VAR_OUTPUT
	OUT_Error				: BOOL;
	OUT_Busy				: BOOL;
END_VAR

VAR
	ETAPE					: UINT;

    myStruct      			: ARRAY[1..CstNbLigneBuffer] OF St_DataHisto;
	myStructMax    			: ARRAY[1..CstNbLigneBufferMax] OF St_DataHisto;
	StructNull				: St_DataHisto;

    SQLDatabase				: FB_SQLDatabaseEvt('',T#10S);
	SQLCommand1				: FB_SQLCommandEvt('',T#10S);
	SQLCommandNull			: FB_SQLCommandEvt('',T#10S);
	bConnected				: BOOL;              	        	

	TrameValues				: T_MaxString := ' ([Timestamp],[Timestamp_Ms],[ParentId],[Value])';
	pPosRequete				: DINT;                		
	RequeteFinale			: ARRAY[1..100] OF STRING(1000);	
	RequeteFinaleNull		: ARRAY[1..100] OF STRING(1000);	
	sTimeStamp				: STRING(255);               	
	RequeteEntete			: STRING(1000);
	sInsertValue			: STRING(1000);
	Format					: FB_FormatString;
	                		
	NbElemBuffer			: DINT;
	KK						: DINT;
	                    	
	CmdStart				: BOOL;
	TrigCmdExec				: R_TRIG;
	TrigStart				: R_TRIG;
	RsStart					: RS;
	
	// Insert
		hDBID_BaseTampon	: UINT := 3;
	// AlarmManagement      
		bBufferMaxFull 		: BOOL;        		
		bInStructNull		: BOOL;
		
		
		
	
END_VAR

NbElemBuffer := M_Count();
CmdStart := NbElemBuffer>= CstNbLigneBuffer;


TrigStart(CLK := CmdStart);
IF TrigStart.Q THEN
	FOR KK := 1 TO CstNbLigneBuffer DO
		myStruct[KK] := myStructMax[KK];
	END_FOR
END_IF


// call functionblock

CASE ETAPE OF
	0://INITIALISATION  & CONNECTION
		RequeteEntete := concat(concat('INSERT INTO ',NomTable),concat(TrameValues,' VALUES '));
		RsStart(SET := TrigStart.Q);
		IF RsStart.Q1 THEN
			IF SQLDatabase.Connect(hDBID := hDBID) THEN;
				bConnected := NOT sqldatabase.bError;
				IF bConnected THEN
					ETAPE := 1;
				ELSE
					ETAPE := 255;
				END_IF
			END_IF
		END_IF
		
	1: // CONNECTED
		IF SQLDatabase.CreateCmd(pSQLCommand := ADR(SQLCommand1)) THEN 
			IF NOT SQLCommand1.bError THEN
				ETAPE := 2;
			ELSIF SQLCommand1.bError THEN
				ETAPE := 255;
			END_IF
		END_IF
	2:
		MEMCPY(srcAddr:= ADR(RequeteEntete), destAddr := ADR(requeteFinale), n:= SIZEOF(RequeteEntete));
		pPosRequete := LEN(STR := RequeteEntete);
		FOR KK:= 1 TO CstNbLigneBuffer-1 DO
			sTimeStamp	:= right(STR := DT_TO_STRING(myStruct[KK].Timestamp), SIZE := LEN(DT_TO_STRING(myStruct[KK].Timestamp))-3);
			Format(sFormat := '($'%s $',%.3d,%.4d,%5.2f),', arg1 := F_STRING(sTimeStamp),arg2:=F_DINT(myStruct[KK].Timestamp_Ms), arg3:= F_DINT(myStruct[KK].ParentId), arg4:= F_LREAL(myStruct[KK].Value), sOut=>sInsertValue);
			MEMCPY(srcAddr:= ADR(sInsertValue), destAddr := ADR(requeteFinale)+DINT_TO_DWORD(pPosRequete), n:= SIZEOF(sInsertValue));
			pPosRequete:= pPosRequete + LEN(STR := sInsertValue);
		END_FOR
		sTimeStamp	:= right(STR := DT_TO_STRING(myStruct[KK].Timestamp), SIZE := LEN(DT_TO_STRING(myStruct[KK].Timestamp))-3);
		Format(sFormat := '($'%s $',%.3d,%.4d,%5.2f)', arg1 := F_STRING(sTimeStamp),arg2:=F_DINT(myStruct[KK].Timestamp_Ms), arg3:= F_DINT(myStruct[KK].ParentId), arg4:= F_LREAL(myStruct[KK].Value), sOut=>sInsertValue);
		MEMCPY(srcAddr:= ADR(sInsertValue), destAddr := ADR(requeteFinale)+DINT_TO_DWORD(pPosRequete), n:= SIZEOF(sInsertValue));
	
		IF SQLCommand1.Execute(pSQLCmd := ADR(RequeteFinale), cbSQLCmd := SIZEOF(Requetefinale))THEN
			
			IF  NOT SQLCommand1.bError THEN
				ETAPE := 3;
			ELSIF SQLCommand1.bError THEN
				ETAPE := 255;
			END_IF
		END_IF
	3:
			IF SQLDatabase.Disconnect() THEN
				ETAPE := 4;
			END_IF 
	4:
		IF NOT SQLDatabase.bError THEN
			RequeteFinale := RequeteFinaleNull;
			FOR KK := CstNbLigneBuffer TO CstNbLigneBufferMax -1 DO
				myStructMax[KK+1-CstNbLigneBuffer]:= myStructMax[KK+1];
			END_FOR
			
			FOR KK := CstNbLigneBufferMax-CstNbLigneBuffer+1 TO CstNbLigneBufferMax DO
				myStructMax[KK]:= StructNull;
			END_FOR			
			
			TrigStart(CLK := FALSE);
			RsStart(RESET1 := TRUE);
			RsStart(RESET1 := FALSE);
			TrigCmdExec(CLK := FALSE);
			CmdStart := FALSE;
			Etape := 0;
			OUT_Error := FALSE;
		ELSE 
			ETAPE := 255;
		END_IF
	255: 
		RequeteFinale := RequeteFinaleNull;
		OUT_Error := TRUE;
		Etape := 0;
		RsStart(RESET1 := TRUE);
		RsStart(RESET1 := FALSE);
		TrigCmdExec(CLK := FALSE);
		CmdStart := FALSE;
		
END_CASE

METHOD M_AddLine : BOOL
VAR_INPUT
	InStruct			: St_DataHisto;
END_VAR

VAR
END_VAR
// Check the biggest buffer isn't full
IF MEMCMP(pBuf1 := ADR(StructNull), pBuf2 := ADR(myStructMax[CstNbLigneBufferMax]), n := SIZEOF(StructNull)) <> 0 THEN
	bBufferMaxFull := TRUE;
ELSE
	//Check the input struct isn't null
	IF MEMCMP(pBuf1 := ADR(StructNull), pBuf2 := ADR(InStruct), n := SIZEOF(StructNull)) = 0 THEN
		bInStructNull := TRUE;
	ELSE
		// We parse the biggest buffer
		FOR KK := 1 TO CstNbLigneBufferMax DO 
			IF MEMCMP(pBuf1 := ADR(StructNull), pBuf2 := ADR(myStructMax[KK]), n := SIZEOF(StructNull)) = 0 THEN
				myStructMax[KK] := InStruct;
				bBufferMaxFull := FALSE;
				EXIT;
			END_IF
		END_FOR
	END_IF
END_IF
END_METHOD

METHOD M_AlarmManager : BOOL
VAR_INPUT
	AlarmCode : WORD;
	
END_VAR


AlarmCode.0 := bBufferMaxFull;
AlarmCode.1 := bInStructNull;
END_METHOD

METHOD M_Count : DINT
VAR_INPUT
END_VAR
VAR

END_VAR
FOR KK := 1 TO CstNbLigneBufferMax DO 

	IF MEMCMP(pBuf1 := ADR(StructNull), pBuf2 := ADR(myStructMax[KK]), n := SIZEOF(StructNull)) = 0 THEN
		EXIT ;
	END_IF
END_FOR

M_Count := MIN(KK, CstNbLigneBufferMax);
END_METHOD

END_FUNCTION_BLOCK

// ---- 00_FunctionsBlocks/Database/SQLite/SQLite_CreateDb_V2_1.TcPOU
PROGRAM SQLite_CreateDb_V2_1
VAR_INPUT
	IN_ConfigDbActuelle		: ARRAY[0..MAX_CONFIGURATIONS] OF ST_ConfigDB; 
	IN_DbType				: UINT:= 1; // 1:T_DBConfig_SQLite, 2:T_DBConfig_SQLCe
	IN_Dir					: T_MAXSTRING;
	IN_Name					: STRING;
	IN_Start				: BOOL;
	IN_TableName			: STRING;
END_VAR
VAR_IN_OUT
	IN_hDBID         		: UDINT;	
END_VAR
VAR_OUTPUT
	OUT_Error				: BOOL;
	OUT_Busy				: BOOL;
	OUT_Result				: INT;
END_VAR
VAR
	Etape					: UINT;
	
	TrigStart				: R_TRIG;
	RsStart					: RS;
	bCreateTable			: BOOL;
	TrigCreateTable			: R_TRIG;
	RsCreateTable			: RS;
	PLCDBCreateEvt 			: FB_PLCDBCreateEvt(sNetID := '', tTimeout := T#5S);
	SqlLiteConf				: T_DBConfig_SQLite;
	DbFullDirName			: T_MAXSTRING;	
	sExtension				: STRING:= '.db';
	tcMessage    	 		: I_TcMessage;
	
	AX_ColArray				: ARRAY[0..3] OF ST_ColumnInfo;
	
	dBID_Test				: UDINT := 1;
	KK						: UDINT;
	bExisteDeja				: BOOL;	
END_VAR

OUT_Busy := TRUE;
AX_ColArray[0].sName := 'TimeStamp';     	AX_ColArray[0].eType := E_ColumnType.DateTime;   	AX_ColArray[0].nLength := 4;    
AX_ColArray[1].sName := 'TimeStamp_Ms';    	AX_ColArray[1].eType := E_ColumnType.Integer;    	AX_ColArray[1].nLength := 4;
AX_ColArray[2].sName := 'ParentId';   		AX_ColArray[2].eType := E_ColumnType.Integer;   	AX_ColArray[2].nLength := 4;
AX_ColArray[3].sName := 'Value';   			AX_ColArray[3].eType := E_ColumnType.Float;   		AX_ColArray[3].nLength := 8;


IF IN_DbType = 1 THEN
	sExtension := '.db';
ELSIF IN_DbType = 2 THEN
	sExtension := '.sdf';
END_IF

DbFullDirName := Concat(STR1:=Concat(STR1:= IN_Dir, STR2 := IN_Name), STR2 := sExtension);
SqlLiteConf.bAuthentification := FALSE;
SqlLiteConf.sServer := DbFullDirName;

FOR KK := 0 TO MAX_CONFIGURATIONS DO
	IF IN_ConfigDbActuelle[KK].sServer = DbFullDirName THEN
		bExisteDeja := TRUE;
		OUT_Result := -1;
		OUT_Busy := FALSE;
		OUT_Error := FALSE;
		bCreateTable := FALSE;
		IN_hDBID := IN_ConfigDbActuelle[KK].hDBID;
		EXIT;
	END_IF
	IF KK = MAX_CONFIGURATIONS THEN
		bExisteDeja := FALSE;
	END_IF
END_FOR

TrigStart(CLK := IN_Start AND NOT bExisteDeja);
RsStart(SET := TrigStart.Q);
IF RsStart.Q1 THEN
	IF PLCDBCreateEvt.Database(pDatabaseConfig := ADR(SqlLiteConf), cbDatabaseConfig := SIZEOF(SqlLiteConf), bCreateXMLConfig := TRUE, pDBID := ADR(dBID_Test)) THEN
		IF PLCDBCreateEvt.ipTcResult.nEventId = 59 THEN
			OUT_Error := FALSE;
			OUT_Result := -1;
			OUT_Busy := FALSE;	
			TrigStart(CLK := FALSE);
			bCreateTable := FALSE;
			Etape := 0;
			RsCreateTable(RESET1 := TRUE);
			RsCreateTable(RESET1 := FALSE);
		ELSIF PLCDBCreateEvt.bError THEN
			tcMessage := PLCDBCreateEvt.ipTcResult;
			OUT_Error := TRUE;
		ELSE
			Etape := 1;
			IN_hDBID := dBID_Test;
			bCreateTable := TRUE; 
		END_IF
		RsStart(RESET1 := TRUE);
		RsStart(RESET1 := FALSE);
	END_IF
END_IF

TrigCreateTable(CLK := bCreateTable);
RsCreateTable(SET:= TrigCreateTable.Q);

IF RsCreateTable.Q1 AND ETAPE = 1 THEN
	IF PLCDBCreateEvt.Table(hDBID := IN_hDBID, sTableName := IN_TableName,  pTableCfg := ADR(AX_ColArray), cbTableCfg := SIZEOF(AX_ColArray)  ) THEN
		IF PLCDBCreateEvt.bError THEN
			Etape := 255;
			OUT_Error := TRUE;
			OUT_Result := -2;
		ELSE
			IN_Start := FALSE;
			bCreateTable := FALSE;
			Etape := 0;
			OUT_Result := 1;
			RsCreateTable(RESET1 := TRUE);
			RsCreateTable(RESET1 := FALSE);
			TrigStart(CLK := False);
			OUT_Busy := FALSE;	
			OUT_Error := FALSE;
		END_IF
	END_IF
END_IF

IF Etape = 255 THEN
	Etape := 0;
	bCreateTable := FALSE;
	IN_Start := FALSE;
	OUT_Busy := FALSE;	
	RsCreateTable(RESET1 := TRUE);
	RsCreateTable(RESET1 := FALSE);
	
END_IF

END_PROGRAM

// ---- 00_FunctionsBlocks/Database/SQLite/SQLite_DeleteConfDb_1.TcPOU
PROGRAM SQLite_DeleteConfDb_1
VAR_INPUT
	IN_DbType				: UINT:= 1; // 1:T_DBConfig_SQLite, 2:T_DBConfig_SQLCe
	IN_hDBID         		: UDINT;
	IN_Start				: BOOL;
	
END_VAR
VAR_OUTPUT
	OUT_Error				: BOOL;
	OUT_Busy				: BOOL;
END_VAR
VAR
	Etape					: UINT;
	
	TrigStart				: R_TRIG;
	RsStart					: RS;
	bDeleteTable			: BOOL;
	TrigDeleteFile			: R_TRIG;
	RsDeleteTable			: RS;
	fbConfigTcDBSrv   		: FB_ConfigTcDBSrvEvt (sNetID := '', tTimeout := T#5S);
	DbFullDirName			: T_MAXSTRING;	
	sExtension				: STRING:= '.db';
	tcMessage    	 		: I_TcMessage;
	
	

END_VAR

OUT_Busy := TRUE;

TrigStart(CLK := IN_Start);
RsStart(SET := TrigStart.Q);
IF RsStart.Q1 THEN
	IF fbConfigTcDBSrv.Delete(eTcDBSrvConfigType := E_TcDBSrvConfigType.Database, hConfigID := IN_hDBID) THEN
		IF fbConfigTcDBSrv.bError THEN
			tcMessage := fbConfigTcDBSrv.ipTcResult;
			OUT_Error := TRUE;
			OUT_Busy := FALSE;
			Etape := 255;
		ELSE 
			OUT_Busy := FALSE;
			OUT_Error := FALSE;
			Etape := 0;
		END_IF
		TrigStart(CLK := FALSE);
		RsStart(RESET1 := TRUE);
		RsStart(RESET1 := FALSE);
	END_IF
END_IF

IF Etape = 255 THEN
	Etape := 0;
	bDeleteTable := FALSE;
	IN_Start := FALSE;
	OUT_Busy := FALSE;	
	RsDeleteTable(RESET1 := TRUE);
	RsDeleteTable(RESET1 := FALSE);
	
END_IF

END_PROGRAM

// ---- 00_FunctionsBlocks/Database/UnixTimestamp.TcPOU
FUNCTION_BLOCK UnixTimestamp
VAR_OUTPUT
    seconds: ULINT;
    milliseconds: ULINT;
END_VAR

VAR
    localSystemTime : FB_LocalSystemTime := ( bEnable := TRUE, dwCycle := 1 );
    getTimeZoneInformation : FB_GetTimeZoneInformation;
    timeZoneInformation : ST_TimeZoneInformation;
    specificLocalTimeToFileTime : FB_TzSpecificLocalTimeToFileTime;
    fileTime: T_FILETIME;
    onZerothSecondLastCycle : BOOL;
END_VAR

// Get local system time
localSystemTime();

// On the zeroth second of each minutesync timezone information
IF (timeZoneInformation.standardName = '' OR (localSystemTime.systemTime.wSecond = 0 AND NOT onZerothSecondLastCycle)) THEN
    getTimeZoneInformation(sNetID := '', bExecute := TRUE, tzInfo => timeZoneInformation);
END_IF;

// Convert local system time to unix timestamps
specificLocalTimeToFileTime(in := Tc2_Utilities.SYSTEMTIME_TO_FILETIME(localSystemTime.systemTime), tzInfo := timeZoneInformation, out => fileTime);
seconds := (SHL(DWORD_TO_ULINT(fileTime.dwHighDateTime), 32) + DWORD_TO_ULINT(fileTime.dwLowDateTime)) / 10000000 - 11644473600;
milliseconds := (SHL(DWORD_TO_ULINT(fileTime.dwHighDateTime), 32) + DWORD_TO_ULINT(fileTime.dwLowDateTime)) / 10000 - 11644473600000;

onZerothSecondLastCycle := localSystemTime.systemTime.wSecond = 0;

END_FUNCTION_BLOCK

// ---- 00_FunctionsBlocks/DataProcessing/Compress/FB_CompressFile.TcPOU
FUNCTION_BLOCK FB_CompressFile
// FB to Compress all files of the directory. 
VAR_INPUT
	IN_Directory			: T_MaxString; // directory of the file to compress
END_VAR
VAR_OUTPUT
END_VAR
VAR
	StartProcess 			: NT_StartProcess;
	bTest 					: BOOL;
	TrigJour				: R_TRIG;
	RsJour					: RS;
	DirAlarms				: T_MaxString;
	DirRawdata				: T_MaxString;
	TimeStructYesterday		: TIMESTRUCT;
END_VAR


TrigJour(CLK := CalLocalTimeStruct.wHour =0);
RsJour(SET := TrigJour.Q);

TimeStructYesterday := DT_TO_SYSTEMTIME( SYSTEMTIME_TO_DT (CalLocalTimeStruct) - T#1D);

IF RsJour.Q1 THEN
	DirAlarms := CONCAT(STR1 := CONCAT(STR1 := CONCAT(STR1 := CONCAT(STR1 := CONCAT(STR1 := CONCAT(STR1 := CONCAT(STR1 := CONCAT(STR1 := CONCAT(STR1 := Concat(STR1 := Concat(STR1 := IN_Directory, STR2 := WORD_TO_STRING(TimeStructYesterday.wYear)), STR2 := '\'), STR2 := WORD_TO_STRING(TimeStructYesterday.wMonth)), STR2 := '\'), STR2:='ALARMS_'), STR2:= WORD_TO_STRING(TimeStructYesterday.wYear)), STR2:='-'),STR2:=WORD_TO_STRING(TimeStructYesterday.wMonth)),STR2:='-'),STR2:=WORD_TO_STRING(TimeStructYesterday.wDay)),STR2:='.csv');
	DirRawdata:= CONCAT(STR1 := CONCAT(STR1 := CONCAT(STR1 := CONCAT(STR1 := CONCAT(STR1 := CONCAT(STR1 := CONCAT(STR1 := CONCAT(STR1 := CONCAT(STR1 := Concat(STR1 := Concat(STR1 := IN_Directory, STR2 := WORD_TO_STRING(TimeStructYesterday.wYear)), STR2 := '\'), STR2 := WORD_TO_STRING(TimeStructYesterday.wMonth)), STR2 := '\'), STR2:='RAWDATA_'), STR2:= WORD_TO_STRING(TimeStructYesterday.wYear)), STR2:='-'),STR2:=WORD_TO_STRING(TimeStructYesterday.wMonth)),STR2:='-'),STR2:=WORD_TO_STRING(TimeStructYesterday.wDay)),STR2:='.csv');
	StartProcess
	(
		NETID := '',
		PATHSTR := 'C:\Windows\System32\compact.exe',
		DIRNAME := 'C:\Windows\System32',
		COMNDLINE :=  CONCAT(STR1:=CONCAT(STR1:=CONCAT(STR1:=CONCAT(STR1:=' /c "',STR2:=DirAlarms), str2:='"  "'), STR2:=DirRawdata),str2:='"'),
		Start := RsJour.Q1,
		TMOUT := T#3M
	);
	IF NOT StartProcess.BUSY THEN
		IF NOT StartProcess.ERR THEN
			StartProcess(Start := FALSE);
			RsJour(RESET1:= TRUE);
			RsJour(RESET1:= FALSE);
		ELSE
			StartProcess(Start := FALSE);
		END_IF
	END_IF	
END_IF

END_FUNCTION_BLOCK

// ---- 00_FunctionsBlocks/DataProcessing/Compress/FUN_CompressCSV.TcPOU
PROGRAM FUN_CompressCSV
VAR_INPUT
	InDirectory 		: T_MaxString;
END_VAR
VAR_OUTPUT
END_VAR
VAR
	Directory1		: T_MaxString;
	Directory2		: T_MaxString;
	FB_Time 			: FB_LocalSystemTime;
	CompressFile	: FB_CompressFile;
	PreviousMonth 	: WORD := 12;
	PreviousYear 	: WORD := 2018;
	CalDirectory 	: T_MaxString;
	DirChange		: BOOL;
	bTest 			: BOOL;
	TimeStruct_Local : TIMESTRUCT;
END_VAR

FB_Time(sNetID := '', bEnable := TRUE, dwCycle := 1, dwOpt := 1, tTimeout := T#50MS, systemTime => TimeStruct_Local);
IF FB_TIME.bValid THEN 
	IF PreviousMonth <> TimeStruct_Local.wMonth THEN
		Directory1 := Concat(InDirectory, concat(WORD_TO_STRING(TimeStruct_Local.wYear), '\'));
		
		IF PreviousYear <> TimeStruct_Local.wYear THEN
			Directory1 := Concat(InDirectory, concat(WORD_TO_STRING(TimeStruct_Local.wYear-1), '\'));
			PreviousYear := TimeStruct_Local.wYear;
		END_IF
		
		Directory2 := Concat(Directory1, concat(WORD_TO_STRING(PreviousMonth), '\'));
		PreviousMonth := TimeStruct_Local.wMonth;
		DirChange := TRUE;
	END_IF

	
	IF DirChange THEN	
		bTest := TRUE;
		CompressFile(IN_Directory := Directory2);	
		DirChange := FALSE;
	END_IF
END_IF

END_PROGRAM

// ---- 00_FunctionsBlocks/DataProcessing/Database/DataBase_V2.TcPOU
PROGRAM DataBase_V2
// Cette fois, plutôt qu'1 base avec 3 tables, faire 3 bases par jour (100ms, 1s, 1m)
// Nouvelle architecture : fichiers minute dans le même fichier qu'historisation, les autres dans Database
 
VAR
	ParamBaseDir					: T_MAXString := 'C:\TwinCAT\Functions\Database\SQLite\';
	ParamHistDir					: T_MaxString := 'C:\TwinCAT\Functions\Historisation\';
	
	ParamDbType						: UINT;
	                        		
	DBID_GLOBAL						: ARRAY[1..3] OF UDINT;
	DBID_ToDelete					: ARRAY[1..3] OF UDINT;
	
	bTest							: BOOL;
	
    AX_DirDB						: ARRAY[1..3] OF T_MaxString :=[ParamBaseDir, ParamBaseDir, ParamBaseDir] ;
	                   		
	MesAlarmCode 					: WORD;
	MesWarningCode					: WORD;
	// INIT
		
                            		
	// CheckConfig          		
		bCheckConfig				: BOOL := TRUE;
		TrigCheckConfig				: R_TRIG;
		TrigInit					: F_TRIG;
		RS_CheckConfig				: RS;
		                    		
		ConfigTcDBSrvEvt  			: FB_ConfigTcDBSrvEvt(sNetId := '', tTimeout:=T#5S);
		                    		
		aDBConfig         			: ARRAY[0..MAX_CONFIGURATIONS] OF ST_ConfigDB;
		aAutoGrpConfig    			: ARRAY[0..MAX_CONFIGURATIONS] OF ST_ConfigAutoLogGrp;
		AX_NameBase					: ARRAY[0..MAX_CONFIGURATIONS] OF T_MaxString;
		AX_hDBID					: ARRAY[0..MAX_CONFIGURATIONS] OF BOOL;
		AX_hDBIDNull				: ARRAY[0..MAX_CONFIGURATIONS] OF BOOL;
		                    		
		nDbCount          			: UDINT;
		nAutoGrpCount     			: UDINT;
		tcMessage         			: I_TcMessage;
	
	// DayTrig 
		Trig_CreateFolder			: R_TRIG;
		RS_CreateFolder				: RS;
		RS_CreateDbDay				: RS;
		RS_DeleteConf				: RS;
		RS_DeleteFiles				: RS;
		RS_CompressOldFiles			: RS;
		bDayTrig					: BOOL:= TRUE;
		bCreateDirErr				: BOOL;
		bCreateDbErr				: BOOL;
		bDeleteConfErr				: BOOL;
		bDeleteFileErr				: BOOL;
		bCompressFileErr			: BOOL;
		CreateDir					: FB_CreateDir_V2;
        AX_Name						: ARRAY[1..3] OF STRING;    
		DeleteFile30Days			: FB_DeleteFile;          
		DeleteFile3Days				: FB_DeleteFile;          
		StartProcess 				: NT_StartProcess;
		
	// CreateDb Init        		
		bCreateDb					: BOOL := TRUE;
		DbidCreated					: UDINT := 1;
		DbCreated_Trig				: F_TRIG;
		AX_ColArray					: ARRAY[0..3] OF ST_ColumnInfo;
	                            	
	// One hour has elapsed
		Trig1hour					: R_TRIG;
		Rs1hour						: RS;
		OldDBID						: UDINT := 1;
		bDbCreated					: BOOL;
		bDbDelete					: BOOL;
		sReqCmd						: T_MAXSTRING;
		
	// New day 
		TrigJour					: R_TRIG;
		RsJour						: RS;
		b1jourSpDoing				: BOOL;
		TimeStruct3days				: TIMESTRUCT;
		TimeStruct1month			: TIMESTRUCT;
		Requete						: T_MaxString;
		sTimeStamp1					: STRING(255);
		sTimeStamp2					: STRING(255);
		Format						: FB_FormatString;
	
		
	// Insert	
	SQLExpert_InsertBuffer_1s		: FB_SQLExpert_InsertBuffer;
	SQLExpert_InsertBuffer_1m		: FB_SQLExpert_InsertBuffer;
	SQLExpert_InsertBuffer_100ms	: FB_SQLExpert_InsertBuffer;

	TON_100ms						: TON;
	TON_1m							: TON;
	TON_1s							: TON;
	

	
	bInit 							: BOOL := TRUE;
	KK								: UDINT;
	LL								: UDINT := 1;

	bTest1 							: BOOL;
	bTest2 							: BOOL;
	
END_VAR

// Trigger pour détecter nouvelle journée -> lance un check config + DayTrig pour faire les proc stockées
TrigJour(CLK := CalLocalTimeStruct.wHour = 0);
bCheckConfig := TrigJour.Q;
Trig_CreateFolder(CLK := TrigJour.Q OR binit);
RS_CreateFolder(SET := Trig_CreateFolder.Q);

// Methode pour vérifier la configuration actuellement activée sur front montant de bCheckConfig
M_Checkconfig();

IF NOT bCheckConfig THEN
	M_DayTrig();
END_IF 

IF bInit THEN
	M_Init();
END_IF

M_AlarmManagement();
(*--------------------------------------------------------------------------------------------*)
(*--------------------------------------------------------------------------------------------*)
// ICI JE LANCE LES ADD BUFFER POUR LES 3 TABLES
IF NOT bInit THEN
	SQLExpert_InsertBuffer_100ms(NomTable := 'Table100ms', hDBID := DBID_GLOBAL[1]);
	SQLExpert_InsertBuffer_1s(NomTable := 'Table1s', hDBID := DBID_GLOBAL[2]);
	SQLExpert_InsertBuffer_1m(NomTable := 'Table1m', hDBID := DBID_GLOBAL[3]);
	
	
	TON_100ms(IN := NOT bInit, PT := T#100MS);
	IF TON_100ms.Q THEN
		FOR KK := 1 TO 100 DO
			SQLExpert_InsertBuffer_100ms.M_AddLine(InStruct := GVL_DataBaseStructures.AX_Struct_100ms[KK]);
		END_FOR
		TON_100ms(IN := FALSE);
		TON_100ms(IN := TRUE);
	END_IF
	
	TON_1s(IN := NOT bInit, PT := T#1S);
	IF TON_1s.Q THEN
		FOR KK := 1 TO 1000 DO
			SQLExpert_InsertBuffer_1s.M_AddLine(InStruct := GVL_DataBaseStructures.AX_Struct_1s[KK]);
		END_FOR
		TON_1s(IN := FALSE);
		TON_1s(IN := TRUE);
	END_IF
	
	TON_1m(IN := NOT bInit, PT := T#1M);
	IF TON_1m.Q THEN
		FOR KK := 1 TO 1000 DO
			SQLExpert_InsertBuffer_1m.M_AddLine(InStruct := GVL_DataBaseStructures.AX_Struct_1m[KK]);
		END_FOR
		TON_1m(IN := FALSE);
		TON_1m(IN := TRUE);
	END_IF	

END_IF
(*--------------------------------------------------------------------------------------------*)
(*--------------------------------------------------------------------------------------------*)

METHOD M_AlarmManagement : BOOL
VAR
		FB_AlarmCodeManager : FB_AlarmCodeManager;
END_VAR
FB_AlarmCodeManager
(
	bAlarm1 := bCreateDirErr,
	bAlarm2 := bCreateDbErr,
	bAlarm3 := bDeleteConfErr,
	bAlarm4 := bDeleteFileErr,
	bAlarm5 := bCompressFileErr,
	wAlarmCode => MesAlarmCode
);
END_METHOD

METHOD M_CheckConfig : BOOL
VAR_INPUT
END_VAR
TrigCheckConfig(CLK := bCheckConfig OR binit);
RS_CheckConfig(SET := TrigCheckConfig.Q);
	
IF RS_CheckConfig.Q1 THEN
	IF ConfigTcDBSrvEvt.Read(
		pDBConfig := ADR(aDBConfig), 
		cbDBConfig := SIZEOF(aDBConfig), 
		pAutologGrpConfig := ADR(aAutoGrpConfig),
		cbAutoLogGrpConfig := SIZEOF(aAutoGrpConfig),
		pDBCount := ADR(nDbCount),
		pAutoLogGrpCount := ADR(nAutoGrpCount))
	 THEN
		IF ConfigTcDBSrvEvt.bError THEN
			tcMessage := ConfigTcDBSrvEvt.ipTcResult;
			bCheckConfig := FALSE; 
		ELSE
			bCheckConfig := FALSE; 
			FOR KK := 0 TO MAX_CONFIGURATIONS DO
				AX_hDBID[aDBConfig[KK].hDBID] := aDBConfig[KK].hDBID <> 0;
				AX_NameBase[KK] :=  aDBConfig[KK].sName;
			END_FOR
		END_IF  
		TrigCheckConfig(CLK := FALSE OR binit);
		RS_CheckConfig(RESET1 := TRUE);
		RS_CheckConfig(RESET1 := FALSE);
	END_IF
END_IF
END_METHOD

METHOD M_DayTrig : BOOL
VAR_INPUT
END_VAR
VAR
	DirTemp			: ARRAY[1..3] OF T_MaxString;
	AX_NameTemp		: ARRAY[1..3] OF STRING := ['Table100ms', 'Table1s', 'Table1m']; 	
	Dir30Days		: T_MaxString;
	Dir3Days		: T_MaxString; 	
	Dir3DaysComp1	: T_MaxString; 	
	Dir3DaysComp2	: T_MaxString; 	

	
END_VAR



TimeStruct3days := DT_TO_SYSTEMTIME( SYSTEMTIME_TO_DT (CalLocalTimeStruct) - T#3D);
TimeStruct1month := DT_TO_SYSTEMTIME( SYSTEMTIME_TO_DT (CalLocalTimeStruct) - T#30D);

// D'abord je commence par créer tous les dossiers
IF RS_CreateFolder.Q1 THEN
	DirTemp[1] := ParamHistDir;
	DirTemp[2] := Concat(STR1 := Concat(STR1 := ParamHistDir, STR2 := WORD_TO_STRING(CalLocalTimeStruct.wYear)), STR2 := '\');
	DirTemp[3] := CONCAT(STR1 := CONCAT(STR1 := Concat(STR1 := Concat(STR1 := ParamHistDir, STR2 := WORD_TO_STRING(CalLocalTimeStruct.wYear)), STR2 := '\'), STR2 := WORD_TO_STRING(CalLocalTimeStruct.wMonth)), STR2 := '\');
	
	AX_DirDB[1] := ParamBaseDir;
	AX_DirDB[2] := ParamBaseDir;
	AX_DirDB[3] := DirTemp[3];
	FOR KK := 1 TO 3 DO 
		AX_Name[KK] := CONCAT(STR1 := CONCAT(STR1 := CONCAT(STR1 := CONCAT(STR1 := CONCAT(STR1 := Concat(STR1 := WORD_TO_STRING(CalLocalTimeStruct.wYear), STR2 := ''), STR2 := WORD_TO_STRING(CalLocalTimeStruct.wMonth)), STR2:= ''), STR2:= WORD_TO_STRING(CalLocalTimeStruct.wDay)), STR2:= '_'), STR2:= AX_NameTemp[KK]);
	END_FOR
	
	IF LL < 4 THEN
		CreateDir(InPath := DirTemp[LL], InExe := LL < 4);
		IF NOT CreateDir.OutBusy THEN
			IF CreateDir.OutError AND NOT CreateDir.OutErrorId =1827 (*Dossier existe déjà*) THEN
				CreateDir(InExe := FALSE);
				bCreateDirErr := TRUE;
			ELSE
				bCreateDirErr := FALSE;
				CreateDir(InExe := FALSE);
				LL := LL + 1;
			END_IF
			CreateDir(InPath := DirTemp[LL], InExe := FALSE);
		END_IF
	ELSE
		RS_CreateFolder(RESET1 := TRUE);
		RS_CreateFolder(RESET1 := FALSE);
		RS_CreateDbDay(SET := TRUE);
		RS_CreateDbDay(SET := FALSE);
		LL := 1;
	END_IF
END_IF

// Ensuite je créée les bases 
IF RS_CreateDbDay.Q1 THEN
	IF LL < 4 THEN
		SQLite_CreateDb_V2(IN_DbType := 1, IN_Dir := AX_DirDB[LL],IN_Name := AX_Name[LL], IN_TableName := AX_NameTemp[LL], IN_hDBID := DBID_GLOBAL[LL], IN_Start := bCreateDb, IN_ConfigDbActuelle := aDBConfig);
		IF NOT SQLite_CreateDb_V2.OUT_Busy THEN
			SQLite_CreateDb_V2(IN_Start := FALSE, IN_hDBID := DBID_GLOBAL[LL]);
			IF SQLite_CreateDb_V2.OUT_Error THEN
				SQLite_CreateDb_V2(IN_Start := FALSE, IN_hDBID := DBID_GLOBAL[LL]);
				bCreateDbErr := TRUE;
			ELSE
				SQLite_CreateDb_V2(IN_Start := FALSE, IN_hDBID := DBID_GLOBAL[LL]);
				LL := LL + 1;
				bCreateDbErr := FALSE;
			END_IF
		END_IF
	ELSE
		LL := 1;
		RS_CreateDbDay(RESET1 := TRUE);
		RS_CreateDbDay(RESET1 := FALSE);
		RS_DeleteConf(SET := TRUE AND NOT bInit);
		RS_DeleteConf(SET := FALSE);
		bDayTrig := False;
	END_IF
END_IF

// Ensuite je supprime les vieilles tables de la conf précédente
IF RS_DeleteConf.Q1 THEN
	IF LL < 4 THEN
		DBID_ToDelete[LL] := SEL(DBID_GLOBAL[LL] = LL, LL, LL+3);
		// CELA NE SUPPRIME QUE LES CONFS
		SQLite_DeleteConfDb(IN_DbType := 1, IN_hDBID := DBID_ToDelete[LL], IN_Start := TRUE);
		IF NOT SQLite_DeleteConfDb.OUT_Busy THEN
			IF SQLite_DeleteConfDb.OUT_Error THEN
				SQLite_DeleteConfDb(IN_Start := FALSE);
				bDeleteConfErr := TRUE;
			ELSE
				bDeleteConfErr := FALSE;
				SQLite_DeleteConfDb(IN_Start := FALSE);
				LL := LL + 1;
			END_IF
		END_IF
	ELSE
		LL := 1;
		RS_DeleteConf(RESET1 := TRUE);
		RS_DeleteConf(RESET1 := FALSE);
		RS_DeleteFiles(SET := TRUE);
		RS_DeleteFiles(SET := FALSE);
	END_IF
END_IF

// Et enfin, je supprime les vieux fichiers : plus de 30 jours pour les 1s, plus de 3 jours pour les 100ms
IF RS_DeleteFiles.Q1 THEN
	Dir30Days := CONCAT(STR1:=CONCAT(STR1:=CONCAT(STR1 := CONCAT(STR1 := CONCAT(STR1 := CONCAT(STR1 := CONCAT(STR1 := Concat(STR1 := ParamBaseDir, STR2 := WORD_TO_STRING(TimeStruct1month.wYear)), STR2 := ''), STR2 := WORD_TO_STRING(TimeStruct1month.wMonth)), STR2:= ''), STR2:= WORD_TO_STRING(TimeStruct1month.wDay)), STR2:= '_'), STR2:= AX_NameTemp[LL]), STR2 := '.db');
	Dir3Days := CONCAT(STR1:=CONCAT(STR1:=CONCAT(STR1 := CONCAT(STR1 := CONCAT(STR1 := CONCAT(STR1 := CONCAT(STR1 := Concat(STR1 := ParamBaseDir, STR2 := WORD_TO_STRING(TimeStruct3days.wYear)), STR2 := ''), STR2 := WORD_TO_STRING(TimeStruct3days.wMonth)), STR2:= ''), STR2:= WORD_TO_STRING(TimeStruct3days.wDay)), STR2:= '_'), STR2:= AX_NameTemp[LL]), STR2 := '.db');
	
	DeleteFile30Days(IN_Dir := Dir30Days, IN_Start := TRUE);
	DeleteFile3Days(IN_Dir := Dir3Days, IN_Start := TRUE);
	
	IF NOT DeleteFile3Days.OUT_Busy AND NOT DeleteFile30Days.OUT_Busy AND LL < 2 THEN
		IF NOT DeleteFile30Days.OUT_Error AND NOT DeleteFile3Days.OUT_Error THEN
			LL := LL + 1;
			DeleteFile30Days(IN_Start := FALSE);
			DeleteFile3Days(IN_Start := FALSE);
			bDeleteFileErr := FALSE;
		ELSE
			bDeleteFileErr := TRUE;
			DeleteFile30Days(IN_Start := FALSE);
			DeleteFile3Days(IN_Start := FALSE);
		END_IF
	ELSIF NOT DeleteFile3Days.OUT_Busy AND NOT DeleteFile30Days.OUT_Busy AND LL = 2 THEN
		IF NOT DeleteFile30Days.OUT_Error AND NOT DeleteFile3Days.OUT_Error THEN
			LL := 1;
			bDeleteFileErr := FALSE;
			DeleteFile30Days(IN_Start := FALSE);
			DeleteFile3Days(IN_Start := FALSE);
			RS_DeleteFiles(reset1 := TRUE);
			RS_DeleteFiles(reset1 := FALSE);
			RS_CompressOldFiles(set := TRUE);
			RS_CompressOldFiles(Set := FALSE);
		ELSE
			bDeleteFileErr := TRUE;
			DeleteFile30Days(IN_Start := FALSE);
			DeleteFile3Days(IN_Start := FALSE);
		END_IF
	END_IF
END_IF

IF RS_CompressOldFiles.Q1 THEN
	Dir3DaysComp1 := CONCAT(STR1:=CONCAT(STR1:=CONCAT(STR1 := CONCAT(STR1 := CONCAT(STR1 := CONCAT(STR1 := CONCAT(STR1 := Concat(STR1 := ParamBaseDir, STR2 := WORD_TO_STRING(TimeStruct3days.wYear)), STR2 := ''), STR2 := WORD_TO_STRING(TimeStruct3days.wMonth)), STR2:= ''), STR2:= WORD_TO_STRING(TimeStruct3days.wDay)), STR2:= '_'), STR2:= AX_NameTemp[1]), STR2 := '.db');
	Dir3DaysComp2 := CONCAT(STR1:=CONCAT(STR1:=CONCAT(STR1 := CONCAT(STR1 := CONCAT(STR1 := CONCAT(STR1 := CONCAT(STR1 := Concat(STR1 := ParamBaseDir, STR2 := WORD_TO_STRING(TimeStruct3days.wYear)), STR2 := ''), STR2 := WORD_TO_STRING(TimeStruct3days.wMonth)), STR2:= ''), STR2:= WORD_TO_STRING(TimeStruct3days.wDay)), STR2:= '_'), STR2:= AX_NameTemp[2]), STR2 := '.db');
	StartProcess
	(
		NETID := '',
		PATHSTR := 'C:\Windows\System32\compact.exe',
		DIRNAME := 'C:\Windows\System32',
		COMNDLINE :=  CONCAT(STR1:=CONCAT(STR1:=CONCAT(STR1:=CONCAT(STR1:=' /c "',STR2:=Dir3DaysComp1), str2:='"  "'), STR2:=Dir3DaysComp2),str2:='"'),
		Start := RS_CompressOldFiles.Q1,
		TMOUT := T#3M
	);
	IF NOT StartProcess.BUSY THEN
		IF NOT StartProcess.ERR THEN
			StartProcess(Start := FALSE);
			bCompressFileErr := FALSE;
			RS_CompressOldFiles(RESET1:= TRUE);
			RS_CompressOldFiles(RESET1:= FALSE);
		ELSE
			StartProcess(Start := FALSE);
			bCompressFileErr := TRUE;
		END_IF
	END_IF	
END_IF
END_METHOD

METHOD M_Init : BOOL
VAR_INPUT
END_VAR


bInit := (bCheckConfig) OR (bDayTrig);
END_METHOD

END_PROGRAM

// ---- 00_FunctionsBlocks/DataProcessing/Database/FB_DeleteFile.TcPOU
FUNCTION_BLOCK FB_DeleteFile
VAR_INPUT
	IN_Start				: BOOL;
	IN_Dir					: T_MaxString;
END_VAR
VAR_OUTPUT
	OUT_Error				: BOOL;
	OUT_Busy				: BOOL;
END_VAR
VAR
	
	TrigStart				: R_TRIG;
	RsStart					: RS;
	FileDelete				: FB_FileDelete;
	
	

END_VAR

OUT_Busy := TRUE;

TrigStart(CLK := IN_Start);
FileDelete(sNetId := '', sPathName := IN_Dir, bExecute := TrigStart.Q);

RsStart(SET := TrigStart.Q);
IF RsStart.Q1 THEN
	IF NOT FileDelete.bBusy THEN
		IF FileDelete.bError THEN
			OUT_Error := TRUE;
			OUT_Busy := FALSE;
		ELSE 
			OUT_Error := FALSE;
			OUT_Busy := FALSE;
		END_IF
		TrigStart(CLK := FALSE);
		RsStart(RESET1 := TRUE);
		RsStart(RESET1 := FALSE);
	END_IF
END_IF

END_FUNCTION_BLOCK

// ---- 00_FunctionsBlocks/DataProcessing/Database/FB_SQLExpert_InsertBuffer.TcPOU
FUNCTION_BLOCK FB_SQLExpert_InsertBuffer
// Fonctionnement : Tableau de 2000 structures en input. Dès qu'on atteint 1000 structures remplies, décalage de l'espace mémoire
// pour en 1 temps de cycle pour ne pas perdre de données sur le transfert.
VAR CONSTANT
	CstNbLigneBuffer		: DINT:= 250;
	CstNbLigneBufferMax	 	: DINT:= 5000;

END_VAR

VAR_INPUT
	NomTable				: STRING := 'Table100ms';
	hDBID					: UDINT;
END_VAR

VAR_OUTPUT
	OUT_Error				: BOOL;
	OUT_Busy				: BOOL;
END_VAR

VAR
	ETAPE					: UINT;

    myStruct      			: ARRAY[1..CstNbLigneBuffer] OF St_DataHisto;
	myStructMax    			: ARRAY[1..CstNbLigneBufferMax] OF St_DataHisto;
	StructNull				: St_DataHisto;

    SQLDatabase				: FB_SQLDatabaseEvt('',T#10S);
	SQLCommand1				: FB_SQLCommandEvt('',T#10S);
	SQLCommandNull			: FB_SQLCommandEvt('',T#10S);
	bConnected				: BOOL;              	        	

	TrameValues				: T_MaxString := ' ([Timestamp],[Timestamp_Ms],[ParentId],[Value])';
	pPosRequete				: DINT;                		
	RequeteFinale			: ARRAY[1..100] OF STRING(1000);	
	RequeteFinaleNull		: ARRAY[1..100] OF STRING(1000);	
	sTimeStamp				: STRING(255);               	
	RequeteEntete			: STRING(1000);
	sInsertValue			: STRING(1000);
	Format					: FB_FormatString;
	                		
	NbElemBuffer			: DINT;
	KK						: DINT;
	                    	
	CmdStart				: BOOL;
	TrigCmdExec				: R_TRIG;
	TrigStart				: R_TRIG;
	RsStart					: RS;
	
	// Insert
		hDBID_BaseTampon	: UINT := 3;
	// AlarmManagement      
		bBufferMaxFull 		: BOOL;        		
		bInStructNull		: BOOL;
		
		
		
	
END_VAR

NbElemBuffer := M_Count();
CmdStart := NbElemBuffer>= CstNbLigneBuffer;


TrigStart(CLK := CmdStart);
IF TrigStart.Q THEN
	FOR KK := 1 TO CstNbLigneBuffer DO
		myStruct[KK] := myStructMax[KK];
	END_FOR
END_IF


// call functionblock

CASE ETAPE OF
	0://INITIALISATION  & CONNECTION
		RequeteEntete := concat(concat('INSERT INTO ',NomTable),concat(TrameValues,' VALUES '));
		RsStart(SET := TrigStart.Q);
		IF RsStart.Q1 THEN
			IF SQLDatabase.Connect(hDBID := hDBID) THEN;
				bConnected := NOT sqldatabase.bError;
				IF bConnected THEN
					ETAPE := 1;
				ELSE
					ETAPE := 255;
				END_IF
			END_IF
		END_IF
		
	1: // CONNECTED
		IF SQLDatabase.CreateCmd(pSQLCommand := ADR(SQLCommand1)) THEN 
			IF NOT SQLCommand1.bError THEN
				ETAPE := 2;
			ELSIF SQLCommand1.bError THEN
				ETAPE := 255;
			END_IF
		END_IF
	2:
		MEMCPY(srcAddr:= ADR(RequeteEntete), destAddr := ADR(requeteFinale), n:= SIZEOF(RequeteEntete));
		pPosRequete := LEN(STR := RequeteEntete);
		FOR KK:= 1 TO CstNbLigneBuffer-1 DO
			sTimeStamp	:= right(STR := DT_TO_STRING(myStruct[KK].Timestamp), SIZE := LEN(DT_TO_STRING(myStruct[KK].Timestamp))-3);
			Format(sFormat := '($'%s $',%.3d,%.4d,%5.2f),', arg1 := F_STRING(sTimeStamp),arg2:=F_DINT(myStruct[KK].Timestamp_Ms), arg3:= F_DINT(myStruct[KK].ParentId), arg4:= F_LREAL(myStruct[KK].Value), sOut=>sInsertValue);
			MEMCPY(srcAddr:= ADR(sInsertValue), destAddr := ADR(requeteFinale)+DINT_TO_DWORD(pPosRequete), n:= SIZEOF(sInsertValue));
			pPosRequete:= pPosRequete + LEN(STR := sInsertValue);
		END_FOR
		sTimeStamp	:= right(STR := DT_TO_STRING(myStruct[KK].Timestamp), SIZE := LEN(DT_TO_STRING(myStruct[KK].Timestamp))-3);
		Format(sFormat := '($'%s $',%.3d,%.4d,%5.2f)', arg1 := F_STRING(sTimeStamp),arg2:=F_DINT(myStruct[KK].Timestamp_Ms), arg3:= F_DINT(myStruct[KK].ParentId), arg4:= F_LREAL(myStruct[KK].Value), sOut=>sInsertValue);
		MEMCPY(srcAddr:= ADR(sInsertValue), destAddr := ADR(requeteFinale)+DINT_TO_DWORD(pPosRequete), n:= SIZEOF(sInsertValue));
	
		IF SQLCommand1.Execute(pSQLCmd := ADR(RequeteFinale), cbSQLCmd := SIZEOF(Requetefinale))THEN
			
			IF  NOT SQLCommand1.bError THEN
				ETAPE := 3;
			ELSIF SQLCommand1.bError THEN
				ETAPE := 255;
			END_IF
		END_IF
	3:
			IF SQLDatabase.Disconnect() THEN
				ETAPE := 4;
			END_IF 
	4:
		IF NOT SQLDatabase.bError THEN
			RequeteFinale := RequeteFinaleNull;
			FOR KK := CstNbLigneBuffer TO CstNbLigneBufferMax -1 DO
				myStructMax[KK+1-CstNbLigneBuffer]:= myStructMax[KK+1];
			END_FOR
			
			FOR KK := CstNbLigneBufferMax-CstNbLigneBuffer+1 TO CstNbLigneBufferMax DO
				myStructMax[KK]:= StructNull;
			END_FOR			
			
			TrigStart(CLK := FALSE);
			RsStart(RESET1 := TRUE);
			RsStart(RESET1 := FALSE);
			TrigCmdExec(CLK := FALSE);
			CmdStart := FALSE;
			Etape := 0;
			OUT_Error := FALSE;
		ELSE 
			ETAPE := 255;
		END_IF
	255: 
		RequeteFinale := RequeteFinaleNull;
		OUT_Error := TRUE;
		Etape := 0;
		RsStart(RESET1 := TRUE);
		RsStart(RESET1 := FALSE);
		TrigCmdExec(CLK := FALSE);
		CmdStart := FALSE;
		
END_CASE

METHOD M_AddLine : BOOL
VAR_INPUT
	InStruct			: St_DataHisto;
END_VAR

VAR
END_VAR
// Check the biggest buffer isn't full
IF MEMCMP(pBuf1 := ADR(StructNull), pBuf2 := ADR(myStructMax[CstNbLigneBufferMax]), n := SIZEOF(StructNull)) <> 0 THEN
	bBufferMaxFull := TRUE;
ELSE
	//Check the input struct isn't null
	IF MEMCMP(pBuf1 := ADR(StructNull), pBuf2 := ADR(InStruct), n := SIZEOF(StructNull)) = 0 THEN
		bInStructNull := TRUE;
	ELSE
		// We parse the biggest buffer
		FOR KK := 1 TO CstNbLigneBufferMax DO 
			IF MEMCMP(pBuf1 := ADR(StructNull), pBuf2 := ADR(myStructMax[KK]), n := SIZEOF(StructNull)) = 0 THEN
				myStructMax[KK] := InStruct;
				bBufferMaxFull := FALSE;
				EXIT;
			END_IF
		END_FOR
	END_IF
END_IF
END_METHOD

METHOD M_AlarmManager : BOOL
VAR_INPUT
	AlarmCode : WORD;
	
END_VAR


AlarmCode.0 := bBufferMaxFull;
AlarmCode.1 := bInStructNull;
END_METHOD

METHOD M_Count : DINT
VAR_INPUT
END_VAR
VAR

END_VAR
FOR KK := 1 TO CstNbLigneBufferMax DO 

	IF MEMCMP(pBuf1 := ADR(StructNull), pBuf2 := ADR(myStructMax[KK]), n := SIZEOF(StructNull)) = 0 THEN
		EXIT ;
	END_IF
END_FOR

M_Count := MIN(KK, CstNbLigneBufferMax);
END_METHOD

END_FUNCTION_BLOCK

// ---- 00_FunctionsBlocks/DataProcessing/Database/SQLite_CreateDb_V2.TcPOU
PROGRAM SQLite_CreateDb_V2
VAR_INPUT
	IN_ConfigDbActuelle		: ARRAY[0..MAX_CONFIGURATIONS] OF ST_ConfigDB; 
	IN_DbType				: UINT:= 1; // 1:T_DBConfig_SQLite, 2:T_DBConfig_SQLCe
	IN_Dir					: T_MAXSTRING;
	IN_Name					: STRING;
	IN_Start				: BOOL;
	IN_TableName			: STRING;
END_VAR
VAR_IN_OUT
	IN_hDBID         		: UDINT;	
END_VAR
VAR_OUTPUT
	OUT_Error				: BOOL;
	OUT_Busy				: BOOL;
	OUT_Result				: INT;
END_VAR
VAR
	Etape					: UINT;
	
	TrigStart				: R_TRIG;
	RsStart					: RS;
	bCreateTable			: BOOL;
	TrigCreateTable			: R_TRIG;
	RsCreateTable			: RS;
	PLCDBCreateEvt 			: FB_PLCDBCreateEvt(sNetID := '', tTimeout := T#5S);
	SqlLiteConf				: T_DBConfig_SQLite;
	DbFullDirName			: T_MAXSTRING;	
	sExtension				: STRING:= '.db';
	tcMessage    	 		: I_TcMessage;
	
	AX_ColArray				: ARRAY[0..3] OF ST_ColumnInfo;
	
	dBID_Test				: UDINT;
	KK						: UDINT;
	bExisteDeja				: BOOL;	
END_VAR

OUT_Busy := TRUE;
AX_ColArray[0].sName := 'TimeStamp';     	AX_ColArray[0].eType := E_ColumnType.DateTime;   	AX_ColArray[0].nLength := 4;    
AX_ColArray[1].sName := 'TimeStamp_Ms';    	AX_ColArray[1].eType := E_ColumnType.Integer;    	AX_ColArray[1].nLength := 4;
AX_ColArray[2].sName := 'ParentId';   		AX_ColArray[2].eType := E_ColumnType.Integer;   	AX_ColArray[2].nLength := 4;
AX_ColArray[3].sName := 'Value';   			AX_ColArray[3].eType := E_ColumnType.Float;   		AX_ColArray[3].nLength := 8;


IF IN_DbType = 1 THEN
	sExtension := '.db';
ELSIF IN_DbType = 2 THEN
	sExtension := '.sdf';
END_IF

DbFullDirName := Concat(STR1:=Concat(STR1:= IN_Dir, STR2 := IN_Name), STR2 := sExtension);
SqlLiteConf.bAuthentification := FALSE;
SqlLiteConf.sServer := DbFullDirName;

FOR KK := 0 TO MAX_CONFIGURATIONS DO
	IF IN_ConfigDbActuelle[KK].sServer = DbFullDirName THEN
		bExisteDeja := TRUE;
		OUT_Result := -1;
		OUT_Busy := FALSE;
		OUT_Error := FALSE;
		bCreateTable := FALSE;
		IN_hDBID := IN_ConfigDbActuelle[KK].hDBID;
		EXIT;
	END_IF
	IF KK = MAX_CONFIGURATIONS THEN
		bExisteDeja := FALSE;
	END_IF
END_FOR

TrigStart(CLK := IN_Start AND NOT bExisteDeja);
RsStart(SET := TrigStart.Q);
IF RsStart.Q1 THEN
	IF PLCDBCreateEvt.Database(pDatabaseConfig := ADR(SqlLiteConf), cbDatabaseConfig := SIZEOF(SqlLiteConf), bCreateXMLConfig := TRUE, pDBID := ADR(dBID_Test)) THEN
		IF PLCDBCreateEvt.ipTcResult.nEventId = 59 THEN
			OUT_Error := FALSE;
			OUT_Result := -1;
			OUT_Busy := FALSE;	
			TrigStart(CLK := FALSE);
			bCreateTable := FALSE;
			Etape := 0;
			RsCreateTable(RESET1 := TRUE);
			RsCreateTable(RESET1 := FALSE);
		ELSIF PLCDBCreateEvt.bError THEN
			tcMessage := PLCDBCreateEvt.ipTcResult;
			OUT_Error := TRUE;
		ELSE
			Etape := 1;
			IN_hDBID := dBID_Test;
			bCreateTable := TRUE; 
		END_IF
		RsStart(RESET1 := TRUE);
		RsStart(RESET1 := FALSE);
	END_IF
END_IF

TrigCreateTable(CLK := bCreateTable);
RsCreateTable(SET:= TrigCreateTable.Q);

IF RsCreateTable.Q1 AND ETAPE = 1 THEN
	IF PLCDBCreateEvt.Table(hDBID := IN_hDBID, sTableName := IN_TableName,  pTableCfg := ADR(AX_ColArray), cbTableCfg := SIZEOF(AX_ColArray)  ) THEN
		IF PLCDBCreateEvt.bError THEN
			Etape := 255;
			OUT_Error := TRUE;
			OUT_Result := -2;
		ELSE
			IN_Start := FALSE;
			bCreateTable := FALSE;
			Etape := 0;
			OUT_Result := 1;
			RsCreateTable(RESET1 := TRUE);
			RsCreateTable(RESET1 := FALSE);
			TrigStart(CLK := False);
			OUT_Busy := FALSE;	
			OUT_Error := FALSE;
		END_IF
	END_IF
END_IF

IF Etape = 255 THEN
	Etape := 0;
	bCreateTable := FALSE;
	IN_Start := FALSE;
	OUT_Busy := FALSE;	
	RsCreateTable(RESET1 := TRUE);
	RsCreateTable(RESET1 := FALSE);
	
END_IF

END_PROGRAM

// ---- 00_FunctionsBlocks/DataProcessing/Database/SQLite_DeleteConfDb.TcPOU
PROGRAM SQLite_DeleteConfDb
VAR_INPUT
	IN_DbType				: UINT:= 1; // 1:T_DBConfig_SQLite, 2:T_DBConfig_SQLCe
	IN_hDBID         		: UDINT;
	IN_Start				: BOOL;
	
END_VAR
VAR_OUTPUT
	OUT_Error				: BOOL;
	OUT_Busy				: BOOL;
END_VAR
VAR
	Etape					: UINT;
	
	TrigStart				: R_TRIG;
	RsStart					: RS;
	bDeleteTable			: BOOL;
	TrigDeleteFile			: R_TRIG;
	RsDeleteTable			: RS;
	fbConfigTcDBSrv   		: FB_ConfigTcDBSrvEvt (sNetID := '', tTimeout := T#5S);
	DbFullDirName			: T_MAXSTRING;	
	sExtension				: STRING:= '.db';
	tcMessage    	 		: I_TcMessage;
	
	

END_VAR

OUT_Busy := TRUE;

TrigStart(CLK := IN_Start);
RsStart(SET := TrigStart.Q);
IF RsStart.Q1 THEN
	IF fbConfigTcDBSrv.Delete(eTcDBSrvConfigType := E_TcDBSrvConfigType.Database, hConfigID := IN_hDBID) THEN
		IF fbConfigTcDBSrv.bError THEN
			tcMessage := fbConfigTcDBSrv.ipTcResult;
			OUT_Error := TRUE;
			OUT_Busy := FALSE;
			Etape := 255;
		ELSE 
			OUT_Busy := FALSE;
			OUT_Error := FALSE;
			Etape := 0;
		END_IF
		TrigStart(CLK := FALSE);
		RsStart(RESET1 := TRUE);
		RsStart(RESET1 := FALSE);
	END_IF
END_IF

IF Etape = 255 THEN
	Etape := 0;
	bDeleteTable := FALSE;
	IN_Start := FALSE;
	OUT_Busy := FALSE;	
	RsDeleteTable(RESET1 := TRUE);
	RsDeleteTable(RESET1 := FALSE);
	
END_IF

END_PROGRAM

// ---- 00_FunctionsBlocks/DataProcessing/FB_Average.TcPOU
FUNCTION_BLOCK  FB_Average
//////////////////
// Calculate the (fixed) Average of a data ( finishing convention )
//////////////////
VAR_INPUT
	ValueIn 			: ANY ; // Value to average
	WindowDuration		: LINT ; // (ms) Window of Time during which the average will be done . 
	
END_VAR
	
VAR_OUTPUT
	ValueOut			: REAL ; // Averaged Value. 
	bError 				: BOOL ; // Switch to true if error i inputs				
END_VAR

VAR
	ValueSum			: REAL ; 							// intermediate Sum value of data in fixed Window range. 
	pAnyReal			: POINTER TO REAL;
	pAnyLReal			: POINTER TO LREAL;
	pAnyULint			: POINTER TO ULINT;
	pAnyUint			: POINTER TO UINT;
	NbPoints			: LINT ; 	// Number of points used for calculating the average. 
	
	JJ					: DINT;		// Pick Up index .
	
END_VAR

// EVALUATE VARIABLES //
NbPoints 		:= WindowDuration 	/ 	CstCycleTime_G  ;  // Number of Cycle in the Window. 
//Ceci est un test pour la subversion. KBT
// CHECK INPUTS //
IF NbPoints =0 THEN 
	bError 		:= TRUE ; 
	ValueOut 	:= -1 ;
	
ELSE
	IF (ValueIn.TypeClass = __SYSTEM.TYPE_CLASS.TYPE_REAL) THEN
		pAnyReal        := ValueIn.pValue; 
		ValueSum  		:= ValueSum + (pAnyReal^);
	ELSIF (ValueIn.TypeClass = __SYSTEM.TYPE_CLASS.TYPE_LREAL) THEN
		pAnyLReal     	:= ValueIn.pValue; 
		ValueSum  		:= ValueSum +  LREAL_TO_REAL(pAnyLReal^);
	ELSIF (ValueIn.TypeClass = __SYSTEM.TYPE_CLASS.TYPE_ULINT) THEN
		pAnyULint     	:= ValueIn.pValue; 
		ValueSum  		:= ValueSum +  ULINT_TO_REAL(pAnyULint^);
	ELSIF (ValueIn.TypeClass = __SYSTEM.TYPE_CLASS.TYPe_uint) THEN
		pAnyUint		:= ValueIn.pValue;
		ValueSum		:= ValueSum + UINT_TO_REAL(pAnyUint^);
	END_IF
	JJ			:=JJ+1 ;
	
	IF JJ =NbPoints THEN  
		ValueOut 	:= ValueSum / LINT_TO_REAL(NbPoints)  ; // Average
		ValueSum 	:= 0 ; 	// Reinitialize sum
		JJ			:= 0 ; // Reinitialize JJ

	END_IF

END_IF

END_FUNCTION_BLOCK

// ---- 00_FunctionsBlocks/DataProcessing/FB_CountBitOfWordAtTrue.TcPOU
FUNCTION_BLOCK FB_CountBitOfWordAtTrue
// Count the number of active bit of a word
VAR_INPUT
	MyWord		 	: WORD;		
END_VAR
VAR_OUTPUT
	NbrBitAtTrue 	: BYTE;
	PosOfLastOne	: BYTE;
END_VAR
VAR
	KK 			 	: BYTE;
	VarTemp		 	: WORD;
END_VAR


NbrBitAtTrue := 0;
FOR KK := 1 TO 16 DO
	Vartemp := ROL(MyWord, KK);
	IF VARtemp.0 THEN
		NbrBitAtTrue := NbrBitAtTrue +1 ;
		PosOfLastOne := KK;
	END_IF
END_FOR

END_FUNCTION_BLOCK

// ---- 00_FunctionsBlocks/DataProcessing/FB_Integrate.TcPOU
FUNCTION_BLOCK FB_Integrate
// This FB increments the value of the Input with every call of the FB. DO NOT CALL THIS TWICE IN A CYCLE.
// Integration is done with the trapeze method
// The Reset input resets the value to 0
VAR_INPUT
	IN_DataToIntegrate		: REAL;
	IN_CmdReset				: BOOL;
	
END_VAR
VAR_OUTPUT
	OUT_IntegrationValue	: REAL;
END_VAR
VAR
	OldData					: REAL;
	OldTime					: TIME;
	DeltaTime				: TIME;
END_VAR

IF OldTime > T#0S THEN
	DeltaTime := TIME()-OldTime;
	
	OUT_IntegrationValue := OUT_IntegrationValue+(IN_DataToIntegrate + OldData)*TIME_TO_REAL(DeltaTime)/2000.0;
	
	OldTime := TIME();
	OldData := IN_DataToIntegrate;
	
	IF IN_CmdReset THEN
		OUT_IntegrationValue := 0.0;
		OldData := 0.0;
	END_IF
ELSE
	OldTime := TIME();
	OldData := IN_DataToIntegrate;
END_IF

END_FUNCTION_BLOCK

// ---- 00_FunctionsBlocks/DataProcessing/FB_MessageDynamique.TcPOU
FUNCTION_BLOCK FB_MessageDynamique
// Allows to create dynamic messages in order to add variable to a string
VAR_INPUT
	
	InMessage	: ST_ValuesAlarms;
	InNbparam	: SINT;
END_VAR
VAR_OUTPUT
	OutMessage	: STRING(150);
END_VAR
VAR
	Valeur  	: STRING(10); // Nom de la balise a tester
	P	    	: INT;		 // Pos de la balise dans une chaine de caractere 
	i,j			: SINT;		// Compteur incrémental
	Temp		: String(150);
END_VAR

Temp:=InMessage.Message;
FOR i:=1 TO InNbparam DO
	IF InMessage.Ax_ParamB[i]<>0 THEN
		Valeur := BOOL_TO_STRING(InMessage.Ax_ParamB[i]^);
		P      := FIND(Temp,concat('<Balise_B',INT_TO_STRING(i)));
		IF P >0 THEN
			Temp:=Replace(Temp,Valeur,10,P);
		ELSE
			EXIT;
		END_IF
	END_IF
END_FOR

FOR j:=1 TO InNbparam DO
	IF InMessage.Ax_ParamI[j]<>0 THEN
		Valeur := SINT_TO_STRING(InMessage.Ax_ParamI[j]^);
		P      := FIND(temp,concat('<Balise_I',INT_TO_STRING(j)));
		IF P >0 THEN
			Temp:=Replace(temp,Valeur,10,P);
		ELSE
			EXIT;
		END_IF
	END_IF
END_FOR
OutMessage:=Temp;

END_FUNCTION_BLOCK

// ---- 00_FunctionsBlocks/DataProcessing/FB_MovingAverage.TcPOU
FUNCTION_BLOCK  FB_MovingAverage
//////////////////
// Calculate the Moving Average of a data. Maximal number of point.
//////////////////

VAR CONSTANT 
	CstNbPointMax			: INT := 1000 ; // Average on one hour, with seconds granularity points

END_VAR


VAR_INPUT
	WindowDuration		: DINT ; // (ms) Window of Time during which the average will be done . 
	ValueIn 			: REAL ; // Value to average
	UpdatePeriod		: DINT ; // (ms) Period at which the value is updated. 
	
END_VAR
	

VAR_OUTPUT
	ValueOut			: REAL ; // Averaged Value. 
	bError 				: BOOL ; // Switch to true if error i inputs				
END_VAR

VAR
	Values 				: ARRAY[1..CstNbPointMax] OF REAL; 	// Value to remove from the average calculation
	
	NbPoints			: DINT ; 	// Number of points used for calculating the average. 
	PointPickUpNb		: DINT ; 	// Number of points to skip in average calculation
	
	JJ					: DINT;		// Pick Up index . 
	KK					: DINT;		// For Loop 
	
END_VAR

// EVALUATE VARIABLES //
PointPickUpNb 	:= UpdatePeriod		/	CstCycleTime_G ;
NbPoints 		:= WindowDuration 	/ 	UpdatePeriod  ;  

// CHECK INPUTS //
IF NbPoints > CstNbPointMax THEN 
	bError 		:= TRUE ; 
	ValueOut 	:= -1 ;
	
ELSE
	// UPDATE VALUE ARRAY WITH NEW VALUE AND REMOVE OLD ONE //
	JJ			:=JJ+1 ;
	
	IF JJ = PointPickUpNb THEN 
		JJ		:= 0 ; // Reinitialize JJ
		
		// Move all values in the array on the right
		FOR KK :=1 TO NbPoints-1 DO 
			Values[NbPoints-KK+1]	:= Values[NbPoints-KK] ;
			
		END_FOR
		
		Values[1] 					:= ValueIn ; 	// Assign first index to new value. 
		
		// CALCULATE AVERAGE // 
			ValueOut 						:= 0 ; 
			
			FOR KK:=1 TO NbPoints DO 
				ValueOut 					:= ValueOut + Values[KK] / DINT_TO_REAL(NbPoints) ; 
			
			END_FOR
		
	END_IF
END_IF

END_FUNCTION_BLOCK

// ---- 00_FunctionsBlocks/DataProcessing/FB_Ramp.TcPOU
FUNCTION_BLOCK FB_Ramp
VAR_INPUT
	IN			: REAL;							(* New Setpoint variable *)
	ASCEND		: REAL;					(* maximum positive slope. Set negative value for no limit *)
	
	DESCEND		: REAL;				(* maximum negative slope (non-negative!!).Set negative value for no limit *)
	TIMEBASE	: TIME;					(* reference for ASCEND/DESCEND :
											t#0s : ASCEND/DESCEND defined per call
											else : ASCEND/DESCEND defined per specified time *)
	IN_RESET_VALUE		: REAL; // Value at which the OUT is reseted 
	RESET				:BOOL;						(* reset *)
END_VAR
VAR_OUTPUT
	OUT								: REAL;						(* output limited by  slope *)
	Out_Completed 					: BOOL ; // True when the ramp is over. 
END_VAR
VAR
	DIFF: REAL;
	OLD_IN: REAL;
	TB,CET:DWORD;
	CLOCK: TON;
	probe:REAL;
END_VAR

Out_Completed := FALSE ;

IF RESET=TRUE OR CLOCK.PT<>TIMEBASE THEN			(* Reset *)
	OUT :=  IN_RESET_VALUE ; 
	OLD_IN:=OUT;
	CLOCK(PT:=TIMEBASE,IN:=FALSE);
	Out_Completed := TRUE  ;
END_IF

DIFF:=IN-OLD_IN;									(* Calculate setpoint difference between old and new setpoint *)

IF TIMEBASE=T#0S THEN								(* PLC Cycletime *)
	IF DIFF>ASCEND AND ASCEND >0 THEN
		OUT:=OLD_IN+ASCEND;
	ELSIF DIFF<-DESCEND AND DESCEND >0 THEN
		OUT:=OLD_IN-DESCEND;
	ELSE
		OUT:=IN;
		Out_Completed := TRUE  ;					// 
	END_IF;
ELSE												(* Slope per timebase *)
	TB:=TIME_TO_DWORD(TIMEBASE);					(* TIMEBASE as DWORD *)
		CLOCK();
	CET:=TIME_TO_DWORD(CLOCK.ET);					(* Elapsed time : correspond to cycle time*)
	IF CET>0 THEN									(* *)
		CLOCK(IN:=FALSE);							(* Restart timer *)
		CLOCK(IN:=TRUE);
		probe:=DIFF*TB/CET;							// SMesIng value difference to fit timebase
		IF probe>ASCEND AND ASCEND >0 THEN						(* ascending *)
			OUT:=OLD_IN+ASCEND*CET/DWORD_TO_REAL(TB);
		ELSIF probe<-DESCEND AND DESCEND >0 THEN					(* descending *)
			OUT:=OLD_IN-DESCEND*CET/DWORD_TO_REAL(TB);
		ELSE										(* If value between max descend and max ascend.  *)
			OUT:=IN;
			Out_Completed := TRUE  ;
		END_IF;
	ELSE											(* keine Zeit verstrichen *)
		CLOCK.PT:=TIMEBASE;							(* => ggf. Initialisierung *)
		CLOCK(IN:=TRUE);							(* => ggf. Timer neu starten *)
		Out_Completed := TRUE  ;
	END_IF;
END_IF;

OLD_IN:=OUT;

END_FUNCTION_BLOCK

// ---- 00_FunctionsBlocks/DataProcessing/FB_Ramp_Time.TcPOU
FUNCTION_BLOCK FB_Ramp_Time
// Y := Ax + B while bStart is set
// Works with time : You can set a max time, and a duration of the ramp :
// if pause is True, the Y value freezes until pause goes to False
// if max time is reached, the Y value goes to the value at maxtime

VAR_INPUT
	A 								: REAL ;	// Slope of the ramp
	B 								: REAL ;	// Initial value of the ramp
	bStart 							: BOOL ;	// Rising edge detection to start the ramp, if false, the ramp stops
	bPause							: BOOL ; 	// Pause signal : the value stop, then continues when bPause goes to false
	RampTime						: TIME ;	// Duration of the ramp
	MaxRampTime						: TIME ; 	// Maximum duration of the ramp (including breaks)
END_VAR                 			

VAR_OUTPUT              			
	Y 								: REAL;
	OutCompleted					: BOOL; 	// Rising edge detection to indicate the ramp is done
END_VAR                 		
	
VAR                     			
	TimeStart 						: TIME;
	TimeDurationPause 				: TIME;
	TimeOnGoing						: TIME;
	TimePauseold					: TIME;
	
	Trig_Start						: R_TRIG;
	Trig_Stop						: F_TRIG;
	Trig_PauseStart					: R_TRIG;
    Trig_OutCompleted				: R_TRIG;
            			
	Real_TimeSinceInit 				: REAL;
	                    	
	RS_TimerOn						: RS;
	TP_RampMaxTime					: TP;
END_VAR

Trig_Start(CLK := bStart);
TP_RampMaxTime(IN := Trig_Start.Q, PT := MaxRampTime);


//Trig_Stop(Clk := bStart AND TP_RampMaxTime.Q );
Trig_PauseStart(CLK := bPause);
Trig_OutCompleted(CLK := RS_TimerOn.Q1 AND TimeOnGoing = RampTime);

RS_TimerOn(SET := Trig_Start.Q, RESET1 := TimeOnGoing = RampTime OR Trig_Stop.Q OR Trig_OutCompleted.Q);


OutCompleted := Trig_OutCompleted.Q;
IF Trig_Start.Q THEN
	TimeStart := TIME();
	TimeDurationPause := T#0S;
	TimePauseOld := T#0S;
END_IF

IF Trig_PauseStart.Q THEN
	TimePauseOld := TIME();
END_IF

IF Trig_OutCompleted.Q THEN
	Trig_OutCompleted(CLK := FALSE);
	TimeOnGoing := T#0S;
END_IF

IF bPause THEN
	TimeDurationPause := TimeDurationPause + TIME() - TimePauseOld;
	TimePauseOld := TIME();
END_IF

IF RS_TimerOn.Q1 THEN
	TimeOnGoing := TIME() - TimeStart - TimeDurationPause;
	Real_TimeSinceInit := TIME_TO_REAL(TimeOnGoing);
	IF TimeStart > T#0S THEN
		Y := B + A * (Real_TimeSinceInit);
	END_IF
END_IF

END_FUNCTION_BLOCK

// ---- 00_FunctionsBlocks/DataProcessing/FB_Smooth.TcPOU
FUNCTION_BLOCK FB_Smooth
////////////////// 
// Smooth Variable Change.
//////////////////	

VAR_INPUT
	Setpoint 		: REAL	:=0.0; 		// Setpoint variable
	Slope 			: REAL	:=5.0; 		// Slope in % of Range per seconds
	DeadBand 		: REAL 	:=2; 		// Deadband in % of Range
	Range 			: REAL; 			// Scale in which the value can evolve 
	CycleTime 		: REAL 	:= 1.0 ; 	// Cycle Time in ms.
	InitialValue 	: REAL ; 			// Initial Value of Slope after Reset
	
	Reset 			: BOOL ; 			// Reset initial Value at rising edge
	
END_VAR

VAR_OUTPUT
	OutValue 		: REAL; 			// Output Value
	
END_VAR

VAR 
	TP_Reset 		: TP;				// Maintain reset for 3 seconds
	
	InValue 		: REAL:=0.0 ; 		//  Input Value
 
END_VAR

// RESET //
	TP_Reset(IN := Reset, PT := T#3S);
	
	IF TP_Reset.Q THEN 
		InValue := InitialValue;
		
	END_IF



// RAMP UP //
	IF (Setpoint<(InValue + DeadBand/100*Range)) AND (SetPoint > (InValue-DeadBand/100*Range)) THEN
		// IF values is inside setpoint deadband 
		OutValue :=SetPoint ; 
		
	ELSIF Setpoint > InValue THEN
		// If value is under setpoint value
		OutValue := MIN(InValue + Slope/100*Range * CycleTime/1000, SetPoint) ; 
		
	ELSE
		// If value is above setpoint value
		OutValue := MAX(InValue - Slope/100*Range * CycleTime/1000, SetPoint) ; 	
		
	END_IF

InValue :=OutValue ;

END_FUNCTION_BLOCK

// ---- 00_FunctionsBlocks/DataProcessing/FUN_Transpose.TcPOU
PROGRAM FUN_Transpose
// Allows to transpose an array 
VAR_INPUT
	In_Array					: ARRAY[1..500] OF ARRAY[1..5] OF STRING;
END_VAR
VAR_OUTPUT
	Out_Array					: ARRAY[1..5] OF ARRAY[1..500] OF STRING;
END_VAR


VAR
	KK: INT;
	LL: INT;
END_VAR

FOR LL := 1 TO 5 DO 
	FOR KK := 1 TO 500 DO
	
		Out_Array[LL][KK] := In_Array[KK][LL];
		
	END_FOR
END_FOR

END_PROGRAM

// ---- 00_FunctionsBlocks/DataProcessing/MergeWord/FB_ISKRA_T5.TcPOU
FUNCTION_BLOCK FB_ISKRA_T5
// FB Utilisée uniquement pour motherfucking ISKRA de mes couilles.... 
// 
VAR_INPUT

	WORD_WEAK		: WORD;				// Strong Word. Word to consider if size equals 1.
	WORD_STRONG		: WORD;
END_VAR
VAR_OUTPUT
	VAR_OUT			: REAL;
END_VAR
VAR
	FullWord		: DWORD;
	ValExp			: SINT;
	ValCorps		: UDINT;
END_VAR


FullWord := SHL(WORD_TO_DWORD(WORD_STRONG), 16) OR WORD_Weak;

ValExp := BYTE_TO_SINT(DWORD_TO_BYTE(SHR(FullWord, 24)));
ValCorps := DWORD_TO_UDINT(SHR(SHL(FullWord, 8),8));

VAR_OUT :=  ValCorps*EXPT(10, ValExp);

END_FUNCTION_BLOCK

// ---- 00_FunctionsBlocks/DataProcessing/MergeWord/FB_ISKRA_T6.TcPOU
FUNCTION_BLOCK FB_ISKRA_T6
// FB Utilisée uniquement pour motherfucking ISKRA de mes couilles.... 
// 
VAR_INPUT

	WORD_WEAK		: WORD;				// Strong Word. Word to consider if size equals 1.
	WORD_STRONG		: WORD;
END_VAR
VAR_OUTPUT
	VAR_OUT			: REAL;
END_VAR
VAR
	
	Filtre			: DWORD := 2#11111111000000000000000000000000;
	FullWord		: DWORD;
	ValExp			: SINT;
	ValCorps		: DINT;
	
END_VAR


FullWord := SHL(WORD_TO_DWORD(WORD_STRONG), 16) OR WORD_Weak;

ValExp := BYTE_TO_SINT(DWORD_TO_BYTE(SHR(FullWord, 24)));

ValCorps := -DWORD_TO_DINT(NOT (FullWord OR Filtre) + 1);


VAR_OUT :=  ValCorps*EXPT(10, ValExp);

END_FUNCTION_BLOCK

// ---- 00_FunctionsBlocks/DataProcessing/MergeWord/FB_MergeWordsToDint.TcPOU
FUNCTION_BLOCK FB_MergeWordsToDint
////////////////// 
// Merge two words or one word into a DINT or UDINT with big endian coding. And finally Output a Real. 
//////////////////	

VAR_IN_OUT
	VAR_OUT 		: REAL ; 	
	
END_VAR

VAR_INPUT
	WORD_STRONG 	: WORD; 			// Strong Word. Word to consider if size equals 1.
	WORD_WEAK 		: WORD 	:= 0; 		// Weak Word. 
	
	SIZE 			: INT	:=1 ; 		// Nomber of words to considers. SIZE is equals to one (defaut) or two
	FIX 			: INT 	:=0 ; 		// Number of decimals (defaut 0)
	
	SIGNED 			: BOOL	:=FALSE; 	// Is the data signed or not (defaut) ? 
	SmaDevice 		: BOOL 	:= FALSE ; 	// True if device is SMA. 

END_VAR

VAR
	VAR_AUX 		: REAL ;			// Temporary variable before applying FIX
END_VAR

// Specific code to SMA 250000TL which provide weird data in case of no power on AC or DC Side
IF SmaDevice AND SIGNED AND (WORD_STRONG = 32768 OR WORD_STRONG = 65535)  THEN
		WORD_STRONG := 0 ;
		WORD_WEAK 	:= 0 ;
		
ELSIF SIGNED AND (WORD_STRONG = 32767 AND WORD_WEAK = 65535  )	THEN 	// Digiware 
		WORD_STRONG := 0 ;
		WORD_WEAK 	:= 0 ;

ELSIF WORD_STRONG=65535 AND WORD_WEAK = 65535 AND SIZE=2 AND NOT SIGNED THEN 
		WORD_STRONG := 0 ;
		WORD_WEAK 	:= 0 ;
		
ELSIF WORD_STRONG=65535 AND NOT SIGNED AND SIZE=1 THEN 
	WORD_STRONG := 0 ;

END_IF




IF SIGNED  THEN
	IF SIZE=2 THEN
		VAR_AUX := DINT_TO_REAL(DWORD_TO_DINT(SHL(WORD_TO_DWORD(WORD_STRONG),16) OR WORD_TO_DWORD(WORD_WEAK))) ; 
	ELSE
		VAR_AUX := INT_TO_REAL(WORD_TO_INT(WORD_STRONG)); 
	END_IF
ELSE
	IF SIZE=2 THEN
		VAR_AUX := DWORD_TO_REAL(SHL(WORD_TO_DWORD(WORD_STRONG),16) OR WORD_TO_DWORD(WORD_WEAK)) ;
	ELSE
		VAR_AUX := WORD_TO_REAL((WORD_STRONG));
	END_IF	
END_IF

VAR_OUT := VAR_AUX/(EXPT(10,FIX));

END_FUNCTION_BLOCK

// ---- 00_FunctionsBlocks/DataProcessing/MergeWord/FB_MergeWordsToFloat.TcPOU
FUNCTION_BLOCK FB_MergeWordsToFloat
////////////////// 
// Merge two words into a real with IEEE 754 coding (for float reading). 
//////////////////	
VAR_IN_OUT
	NUMBER_F 		 : REAL;	
END_VAR


VAR_INPUT
	WORD_STRONG_F 	AT %MB82 : WORD; // Strong Word 
	WORD_WEAK_F 	AT %MB80 : WORD; // Weak Word. 
END_VAR

VAR_OUTPUT
	OUT_NanError			: BOOL ; 
END_VAR

VAR
	NUMBER_F_OLD		AT %MB80	: REAL; 	// Works only if the Fb is instantied once per call in the Fb and not the Methods.
	
END_VAR


IF NOT(NUMBER_F_OLD = NUMBER_F_OLD) THEN
	OUT_NanError := TRUE ; 
ELSE
	NUMBER_F :=  NUMBER_F_OLD ; 
	OUT_NanError := FALSE ; 
END_IF

END_FUNCTION_BLOCK

// ---- 00_FunctionsBlocks/DataProcessing/MergeWord/FB_MergeWordsToUint.TcPOU
FUNCTION_BLOCK FB_MergeWordsToUint
////////////////// 
// Merge two words or one word into a DINT or UDINT with big endian coding. And finally Output a Real. 
//////////////////	

VAR_IN_OUT
	VAR_OUT 		: UINT ; 	
	
END_VAR

VAR_INPUT
	WORD_STRONG 		: WORD; 			// Strong Word. Word to consider if size equals 1.
	WORD_WEAK	 		: WORD 	:= 0; 		// Weak Word. 
	

END_VAR

VAR
	VAR_AUX 		: ULINT ;			
	
END_VAR


MEMCPY(destAddr := ADR(VAR_OUT)+1*SIZEOF(WORD_STRONG), 		srcAddr := ADR(WORD_WEAK), 		n := SIZEOF(WORD_WEAK));
MEMCPY(destAddr := ADR(VAR_OUT)+0*SIZEOF(WORD_STRONG), 		srcAddr := ADR(WORD_STRONG), 	n := SIZEOF(WORD_WEAK));

END_FUNCTION_BLOCK

// ---- 00_FunctionsBlocks/DataProcessing/MergeWord/FB_MergeWordsToUlint.TcPOU
FUNCTION_BLOCK FB_MergeWordsToUlint
////////////////// 
// Merge two words or one word into a DINT or UDINT with big endian coding. And finally Output a Real. 
//////////////////	

VAR_IN_OUT
	VAR_OUT 		: ULINT ; 	
	
END_VAR

VAR_INPUT
	WORD1 		: WORD; 			// Strong Word. Word to consider if size equals 1.
	WORD2 		: WORD 	:= 0; 		// Weak Word. 
	WORD3 		: WORD 	:= 0; 		// Weak Word. 
	WORD4 		: WORD 	:= 0; 		// Weak Word. 
	

END_VAR

VAR
	VAR_AUX 		: ULINT ;			
	
END_VAR



MEMCPY(destAddr := ADR(VAR_OUT)+3*SIZEOF(word1), srcAddr := ADR(WORD1), n := SIZEOF(word1));
MEMCPY(destAddr := ADR(VAR_OUT)+2*SIZEOF(word1), srcAddr := ADR(WORD2), n := SIZEOF(word1));
MEMCPY(destAddr := ADR(VAR_OUT)+1*SIZEOF(word1), srcAddr := ADR(WORD3), n := SIZEOF(word1));
MEMCPY(destAddr := ADR(VAR_OUT)+0*SIZEOF(word1), srcAddr := ADR(WORD4), n := SIZEOF(word1));

END_FUNCTION_BLOCK

// ---- 00_FunctionsBlocks/DataProcessing/MergeWord/FB_SplitFloatToWords.TcPOU
FUNCTION_BLOCK FB_SplitFloatToWords
////////////////// 
// Merge two words into a real with IEEE 754 coding (for float reading). 
//////////////////	
VAR_INPUT
	
	VAR_IN 		AT %MD0 : REAL;
END_VAR

VAR_OUTPUT
	
	WORD_STRONG 	AT %MW1 : WORD; // Strong Word 
	WORD_WEAK 	AT %MW0 : WORD; // Weak Word. 
END_VAR

END_FUNCTION_BLOCK

// ---- 00_FunctionsBlocks/DataProcessing/MergeWord/FB_WordsToDint64BE.TcPOU
FUNCTION_BLOCK FB_WordsToDint64BE
////////////////// 
// Merge four words into a DINT or UDINT with big endian coding. And finally Output a Real. 
//////////////////	
VAR_OUTPUT
	OutCalDint : ULINT ; 	
END_VAR

VAR_INPUT
	InFirstWord 		: WORD; 
	InSecondWord 		: WORD; 
	InThirdWord 		: WORD; 
	InFourthWord 		: WORD; 
END_VAR

OutCalDint:= LWORD_TO_ULINT( (SHL(WORD_TO_LWORD(InFirstWord),48) OR SHL(WORD_TO_LWORD(InFirstWord),32)OR SHL(WORD_TO_LWORD(InThirdWord),16)OR WORD_TO_LWORD(InFourthWord)));

END_FUNCTION_BLOCK

// ---- 00_FunctionsBlocks/DataProcessing/MergeWord/FB_WordsToFloat32MLE.TcPOU
FUNCTION_BLOCK FB_WordsToFloat32MLE
////////////////// 
// Merge two words or one word into a Real with Mid little endian coding.
//Validée par KBT : 8/11/2017 
//////////////////		
VAR_INPUT
	
	InFirstWord AT %MW0: WORD; 		// Word sent or stored first 
	InSecondWord AT %MW1 : WORD; 	// Word sent or stored last  

END_VAR
VAR_OUTPUT
	OutCalReal AT %MD0 : REAL;		//Output : Real
END_VAR

END_FUNCTION_BLOCK

// ---- 00_FunctionsBlocks/DataProcessing/ReadFile/FB_ReadCSV.TcPOU
FUNCTION_BLOCK FB_ReadCSV
//Permet de lire les Valeurs de max 1 semaine de points (1 pt/min pdt 7 jours)

VAR_INPUT
	InDirectory_Stockage 		: T_MaxString;		// Base file of the Historization 
	InVariable					: T_MaxString;
	InStartTimeStamp			: TIMESTRUCT;
	InNbLecture					: UINT := 144;
	InExecute					: BOOL;			//Rising Edge detection of read
	ParamSeparateur				: STRING;
	InStructValues				: ARRAY[1..500] OF ST_ValuesWrite;
END_VAR                 		

VAR_OUTPUT              		
	OutValue					: ARRAY[1..10000] OF REAL;
	OutTimeStamp				: ARRAY[1..10000] OF TIMESTRUCT;
	OutCompleted				: BOOL;
	OutbBusy					: BOOL;
	OutError 					: BOOL;
	OutErrorID 					: UINT; // 1 : File not found
END_VAR                 		
VAR     
	// Initialisation 
	CP_READ						: BOOL;
	TypeFile					: STRING;
	ParamTimeOut				: TIME := T#1S;
	
	//Read
	TimeStructBeingRead			: TIMESTRUCT;
	FullDirectory				: STRING;                		
	ReadNewFile					: BOOL;
	
	
	OpenFile					: FB_FileOpen;
	ReadFile					: FB_FileGets;
	CloseFile					: FB_FileClose;
	LineStart					: UINT;			// Ligne de début de la lecture
	LineEnd						: UINT;			// Ligne de fin de la lecture
	LineLeft					: UINT;			// Nombre total de lignes restantes
	Index_Array_OutValue		: UINT;			// Valeur de OutValue qui va être écrite
	
	Opening						: BOOL := TRUE;
	Reading						: BOOL;
	Closing						: BOOL;
	LineRead					: ARRAY[1..20] OF T_Maxstring;
	LineReadNull				: ARRAY[1..20] OF T_Maxstring;
	ColumnNbRead				: UINT;
	TimeStampRead				: STRING(255);
	ValueRead					: STRING(255);
	EOF_Reached					: BOOL;
	PosCursor					: DINT;
                    		
	CompteurLigne				: CTU;
	CompteurLigneRead			: CTU;
	OutBusy						: RS;
	Trig_Read					: R_TRIG;
	Trig_Start 					: R_TRIG;
	
	FileHandle					: UINT;
	FileHandle_Old				: UINT;
	
	NbJours						: UINT;
	KK: UINT 					:= 1;
	bInit 						: BOOL;
	FinalElemStruct				: UINT := 20;
	LL							: UINT := 1;
	LenLineRead					: INT;
END_VAR

IF  Trig_Start.Q THEN
	M_Init();
END_IF

CP_Read := SYSTEMTIME_TO_DT(InStartTimeStamp) + LINT_TO_TIME(InNbLecture*60000) < SYSTEMTIME_TO_DT(CalLocalTimeStruct);
 Trig_Start(CLK := InExecute);
CompteurLigneRead(PV := InNbLecture, RESET := Trig_Start.Q);

OutBusy(Set := CP_Read AND InExecute, RESET1 := OutError OR OutCompleted);
OutbBusy := OutBusy.Q1;

OutCompleted := CompteurLigneRead.Q;

IF OutBusy.Q1 THEN	
	// J'initialise le tout : 
		//Initialisation du type de fichier
			TypeFile := 'RAWDATA'; 
			
		// Calcul du nb de fichiers à ouvrir
			NbJours := DINT_TO_UINT( TRUNC(UINT_TO_INT(InNbLecture + InStartTimeStamp.wHour *60 + InStartTimeStamp.wMinute)/(24*60))+1);

	IF KK <= NbJours THEN
		// Nbre d'heures * 60 + Nbre de minutes + 2 lignes de presentation
		IF KK = 1 THEN
			LineStart := (InStartTimeStamp.wHour *60 + InStartTimeStamp.wMinute + 2); 
			// Calcul des lignes de la lecture : 
			LineLeft := InNbLecture;
		ELSE
			LineStart := 2;
		END_IF
		
		LineEnd := MIN(1442, LineLeft);

		CompteurLigne(PV := LineStart+LineEnd);
		
		TimeStructBeingRead := DT_TO_SYSTEMTIME(SYSTEMTIME_TO_DT(InStartTimeStamp) + LINT_TO_TIME(24*3600000*(KK-1)));
		FullDirectory := Concat(Concat(Concat(Concat(Concat(Concat(Concat(Concat(Concat(Concat(Concat(Concat(InDirectory_Stockage , WORD_TO_STRING(TimeStructBeingRead.wyear)),'\'),WORD_TO_STRING(TimeStructBeingRead.wMonth)),'\'),'RAWDATA'),'_'),WORD_TO_STRING(TimeStructBeingRead.wyear)),'-'),WORD_TO_STRING(TimeStructBeingRead.wMonth)),'-'),WORD_TO_STRING(TimeStructBeingRead.wDay)),'.csv');

		//Ouverture du Fichier, récupération du handle
		OpenFile
		(
			sNetId := '',
			sPathName := FullDirectory,
			nMode := FOPEN_MODEREAD,
			ePath := PATH_GENERIC,
			bExecute := Opening AND NOT OutCompleted,
			hFile => FileHandle
		);
		
		IF OpenFile.nErrId = 1804 THEN // Le fichier n'existe pas 
			OutErrorID := 1;
			OutError := OpenFile.bError;
		ELSIF OpenFile.bError THEN		// Il y a eu une autre erreur
			OutError := OpenFile.bError;
		ELSIF NOT OpenFile.bError AND NOT OpenFile.bBusy AND FileHandle <> 0 AND FileHandle <> FileHandle_Old THEN
			Opening := FALSE;
			FileHandle_Old := FileHandle;
		END_IF
		// On a obtenu le file handle, on va commencer la lecture
		
		
		// Le bloc suivant va lire le document ligne à ligne en incrémentant le compteur ligne et en ressortant l'ensemble de la ligne dans LineRead
		
		IF NOT opening AND NOT CompteurLigneRead.Q AND NOT EOF_Reached THEN		
			IF LL <= 20 THEN
				ReadFile
				(
					sNetId := '',
					hFile := FileHandle,
					bExecute := TRUE,
					tTimeout := ParamTimeOut,
					sLine => LineRead[LL],
					bEOF => EOF_Reached
				);	
				IF NOT ReadFile.bBusy AND NOT ReadFile.bError AND lineread[LL] <> '' THEN
					ReadFile(bExecute := FALSE);
					LenLineRead := LEN(STR := LineRead[LL]);
					IF LenLineRead = 254 THEN
						LL := LL + 1 ;
					ELSE
						FinalElemStruct := LL;
						LL := 1;
					END_IF
				END_IF
			END_IF
			
			IF NOT ReadFile.bBusy AND NOT ReadFile.bError AND (LineRead[FinalElemStruct] <> '' OR EOF_Reached) THEN
				ReadFile(bExecute := FALSE);
				CompteurLigne(CU := TRUE);	
				CompteurLigne(CU := FALSE);
				FinalElemStruct := 20;
				
				IF CompteurLigne.CV >= LineStart + 1 THEN
					TimeStampRead := Substring_Cari
					(
						IN_Delimiter := ParamSeparateur, 
						IN_TextToSearch := LineRead, 
						IN_Position := 0
					);
					OutTimeStamp[Index_Array_OutValue+1]:= FUN_FormatDate(In_String := TimeStampRead);
					
					ValueRead := Substring_Cari
					(
						IN_Delimiter := ParamSeparateur, 
						IN_TextToSearch := LineRead, 
						IN_Position := ColumnNbRead + 1
					);
					OutValue[Index_Array_OutValue+1] := STRING_TO_REAL(ValueRead)*100;
					CompteurLigneRead(CU := TRUE);
					CompteurLigneRead(CU := FALSE);
					Index_Array_OutValue := Index_Array_OutValue + 1;
					
					LL := 1;
				END_IF
				LineRead := LineReadNull;
			ELSIF NOT ReadFile.bBusy AND  ReadFile.bError THEN
				OutError := TRUE;			
			END_IF
		ELSIF EOF_Reached THEN
			ReadFile(bExecute := FALSE);
	
			CloseFile
			(
				sNetId := '',
				bExecute := TRUE,
				hFile := FileHandle,
				tTimeout := ParamTimeOut
			);
			IF NOT CloseFile.bBusy AND NOT CloseFile.bError  THEN
				LineLeft := LineLeft - CompteurLigneRead.CV + 2;
				Index_Array_OutValue := Index_Array_OutValue -1;
				CloseFile(bExecute := FALSE);
				CompteurLigne(RESET := TRUE);
				CompteurLigne(RESET := FALSE);
				Opening := TRUE;
				EOF_Reached := FALSE;
				KK := KK + 1;
			END_IF	
		END_IF
	END_IF
ELSIF EOF_Reached OR CompteurLigneRead.Q AND FileHandle <> 0 THEN
	ReadFile(bExecute := FALSE);
	
	CloseFile
	(
		sNetId := '',
		bExecute := TRUE,
		hFile := FileHandle,
		tTimeout := ParamTimeOut
	);
	IF NOT CloseFile.bBusy AND NOT CloseFile.bError THEN
		CloseFile(bExecute := FALSE);
		CompteurLigne(RESET := TRUE);
		CompteurLigne(RESET := FALSE);
		Opening := TRUE;
		Index_Array_OutValue := 0;
		FileHandle := 0;
		KK := 1;
	ELSIF NOT CloseFile.bBusy AND closefile.bError THEN
		OutError := TRUE;
	END_IF  
END_IF

METHOD M_Init : BOOL
VAR_INPUT
END_VAR

VAR
	KK : UINT;
END_VAR
ColumnNbRead := 1;
FOR KK := 1 TO 500 DO
	IF InVariable = InStructValues[KK].Description THEN
		ColumnNbRead := KK;
		EXIT;
	END_IF
END_FOR
END_METHOD

END_FUNCTION_BLOCK

// ---- 00_FunctionsBlocks/DataProcessing/SavePersistent.TcPOU
PROGRAM SavePersistent
///////////////////
// Save persistent data regularly
///////////////////
VAR
	FB_WritePersistentData : WritePersistentData  ;
	
	LTP2: TP;
	ClockPersistent: BOOL;
END_VAR

// WRITING CLOCK //
	LTP2(IN:=NOT LTP2.Q , PT:= T#1M);
	ClockPersistent := LTP2.Q;

FB_WritePersistentData(
						NETID:='', 
						PORT:= 851 ,
						START :=  ClockPersistent AND NOT FB_WritePersistentData.BUSY , 
						TMOUT := T#10S ) ;

END_PROGRAM

// ---- 00_FunctionsBlocks/DataProcessing/SplitWord/FB_SplitRealToWords.TcPOU
FUNCTION_BLOCK FB_SplitRealToWords
////////////////// 
// Convert one REAL into  2 separate WORDS in Big Endian Encoding. 
//////////////////	
VAR_INPUT
	IN		: REAL ;				// Real input
	
END_VAR

VAR_OUTPUT
	OUT		: ARRAY[0..1]OF WORD;	// Word output array
	
END_VAR

OUT[1] := DWORD_TO_WORD(SHR(SHL(REAL_TO_DWORD(IN),16),16)) ; 	// Strong Word
OUT[0] := DWORD_TO_WORD(SHR(REAL_TO_DWORD(IN),16)); 			// Weak Word

END_FUNCTION_BLOCK

// ---- 00_FunctionsBlocks/DataProcessing/SplitWord/FB_SplitRealToWords_IEEE754.TcPOU
FUNCTION_BLOCK FB_SplitRealToWords_IEEE754
VAR_INPUT
	IN_Real : REAL;
END_VAR
VAR_OUTPUT
	OUT_WordStrong :  WORD;
	OUT_WordWeak :  WORD;

END_VAR
VAR

END_VAR

MEMCPY(destAddr := ADR(OUT_WordStrong), srcAddr := ADR(IN_Real), n := 2);
MEMCPY(destAddr := ADR(OUT_WordWeak), srcAddr := ADR(IN_Real) + 2, n := 2);

END_FUNCTION_BLOCK

// ---- 00_FunctionsBlocks/DataProcessing/SplitWord/FB_SplitUlintToWords.TcPOU
FUNCTION_BLOCK FB_SplitUlintToWords
VAR_INPUT
	IN_ULINT : ULINT;
END_VAR
VAR_OUTPUT
	OUT_WorDS_Transfoong :  WORD;
	OUT_WordWeak :  WORD;

END_VAR
VAR

END_VAR

MEMCPY(destAddr := ADR(OUT_WorDS_Transfoong), srcAddr := ADR(IN_ULINT), n := 2);
MEMCPY(destAddr := ADR(OUT_WordWeak), srcAddr := ADR(IN_ULINT) + 2, n := 2);

END_FUNCTION_BLOCK

// ---- 00_FunctionsBlocks/DataProcessing/SplitWord/FB_SplitWordToByte.TcPOU
FUNCTION_BLOCK FB_SplitWordToByte
////////////////// 
// Convert one REAL into  2 separate WORDS in Big Endian Encoding. 
//////////////////	
VAR_INPUT
	IN		: WORD ;				// Real input
	
END_VAR

VAR_OUTPUT
	STRONG_BYTE		: BYTE;	// Word output array
	WEAK_BYTE		: BYTE;	// Word output array
END_VAR

STRONG_BYTE := WORD_TO_BYTE(IN) ; 				
WEAK_BYTE 	:= WORD_TO_BYTE(SHR(IN,8));

END_FUNCTION_BLOCK

// ---- 00_FunctionsBlocks/DataProcessing/Substring.TcPOU
PROGRAM Substring
// Gives nth occurence of the string encased by delimiter where n = In_Position
//Donne la position de la IN_Position-ième répétition du caractère recherché et renvoie la chaine de caractères suivante
VAR_INPUT
	IN_Delimiter 		: STRING;
	IN_TextToSearch		: T_MaxString;
	IN_Position			: UINT;
END_VAR

VAR
	n					: UINT;	
	Position_Int		: UINT;
	TextToSearch_Int	: T_MaxString;
END_VAR

VAR_OUTPUT
	OUT_NextString			: T_Maxstring;
END_VAR

n:= 0;
TextToSearch_Int := IN_TextToSearch;
Position_Int := INT_TO_UINT( Find(STR1 := TextToSearch_Int, STR2 := IN_Delimiter));


WHILE Position_Int > 0 AND n < IN_Position DO
	OUT_NextString := LEFT(STR := TextToSearch_Int, SIZE := UINT_TO_INT(Position_Int));
	TextToSearch_Int := RIGHT(STR := TextToSearch_Int, SIZE := LEN(STR:= TextToSearch_Int)- LEN(STR := OUT_NextString));
	Position_Int := INT_TO_UINT(FIND(STR1 := TextToSearch_Int, STR2 := IN_Delimiter));
	n := n + 1;
END_WHILE

IF n <> IN_Position THEN
	OUT_NextString := '';
ELSE
	OUT_NextString := left(STR:= OUT_NextString, SIZE := LEN(STR := OUT_NextString) -1);
END_IF

END_PROGRAM

// ---- 00_FunctionsBlocks/DataProcessing/WriteFile/CheckStruct_Alarms.TcPOU
FUNCTION CheckStruct_Alarms : BOOL
//Allows to compare 2 Struct_InputRTU, TRUE if struct are the same
VAR_INPUT
	InStruct1 : ST_ValuesAlarms;
	InStruct2 : ST_ValuesAlarms;
END_VAR
VAR
	bCompareBuffer 	: BOOL := TRUE;
	KK 				: UINT;
END_VAR

CheckStruct_Alarms := InStruct1.Message = Instruct1.Message and InStruct1.ID = Instruct2.ID and InStruct1.Value = InStruct2.Value and InStruct1.Written = Instruct2.Written;

END_FUNCTION

// ---- 00_FunctionsBlocks/DataProcessing/WriteFile/FB_Write_CSV.TcPOU
FUNCTION_BLOCK FB_Write_CSV
VAR_INPUT
	InDirectory 		: T_MaxString;
	AX_StructureValues	: ARRAY[1..500] OF ST_ValuesWrite;
	
	ParamNbColumns		: UINT := 200; 				(* (NA) Number of columns of the file*)
	ParamSeparateur		: STRING := ';';			(* (NA) Separator*)
	ParamDec			: STRING := ',';			(* (NA) ParamDec*)
	ParamExtension		: T_MaxString := '.csv'; 	(* (NA) csv extension *)
END_VAR
VAR_OUTPUT
END_VAR
VAR
	
    CompressFile        : FB_CompressFile;

MesData		: LoggerCSV;
	bWriteAlarm			: BOOL;						// Writing CSV File failed 
	TON_WritealarmFile	: TON;	
	// Data processing 
	format_string		: FB_FormatString;
	AX_AverageFunctions	: ARRAY[1..1000] OF FB_Average;
	AX_AverageValues	: ARRAY[1..1000] OF REAL;
	LenStringToWrite	: INT;
	
	GetHostName			: FB_GetHostName;
	CalFileName			: STRING;
	CalFileName_Old		: STRING;
	CalDate				: STRING;
	CalDate_Old				: STRING;
	
	//Test existence file 

	bFileOK				: BOOL := TRUE ;
	bDirChange			: BOOL;
	FindFile 			: FB_EnumFindFileEntry ;
	FileInfo			: ST_FindFileEntry;
	
	//Initial File creation 
	InitLine			: T_MaxString;
	LastInitLine		: T_MaxString;
	WelcomeMessage 		: T_MaxString := 'Daily rawdata file';
	ForDay				: T_MaxString := 'for day : ';
	ForPlant	 		: T_MaxString := 'for plant : ';
	NewLineVar			: T_MaxString := '$N';
	TimeStampVar		: T_MaxString := 'TimeStamp';
	len_to_write		: INT;
	len_to_add			: INT;
	
	WriteFileInit		: FB_WriteFile;
	WriteFile			: FB_WriteFile;
	MessageInitial		: ARRAY[1..100] OF T_Maxstring;
	MessageInitialNull	: ARRAY[1..100] OF T_Maxstring;
	bInitWrite			: BOOL;
	bInitWriting		: BOOL;
	
	// Write File
	LineToWrite			: ARRAY [1..100] OF  T_Maxstring;
	LineToWrite_Null	: ARRAY [1..100] OF  T_Maxstring;
	ValueToWrite		: T_MaxString;
	TriggerSampling		: R_TRIG;
	
	// General variables
	KK: UINT;
	bInit : BOOL;
	MesTimeStamp : STRING(19);
	

	
END_VAR

M_AlarmManager();
M_DataProcessing ();

IF NOT bInit THEN
	GetHostName(bExecute := FALSE);
	GetHostName(bExecute := TRUE);
	bInit := TRUE;
END_IF

format_string(
	sFormat := 'RAWDATA_%0.2d-%0.2d-%0.2d%s', 
	arg1 := F_WORD(in:=CalLocalTimeStruct.wYear),	arg2 := F_WORD(in:=CalLocalTimeStruct.wMonth),	arg3 := F_WORD(in:=CalLocalTimeStruct.wDay),
	arg4 := F_STRING(in:=ParamExtension),
	sOut => CalFileName
);

format_string(
	sFormat := '%0.2d-%0.2d-%0.2d', 
	arg1 := F_WORD(in:=CalLocalTimeStruct.wYear),	arg2 := F_WORD(in:=CalLocalTimeStruct.wMonth),	arg3 := F_WORD(in:=CalLocalTimeStruct.wDay),
	sOut => CalDate
);

format_string(
	sFormat := '%0.2d-%0.2d-%0.2d %0.2d:%0.2d:%0.2d', 
	arg1 := F_WORD(in:=CalLocalTimeStruct.wYear),	arg2 := F_WORD(in:=CalLocalTimeStruct.wMonth),	arg3 := F_WORD(in:=CalLocalTimeStruct.wDay),
	arg4 := F_WORD(in:=CalLocalTimeStruct.wHour),	arg5 := F_WORD(in:=CalLocalTimeStruct.wMinute),	arg6 := F_WORD(in:=CalLocalTimeStruct.wSecond),
	sOut => MesTimeStamp
);

InitLine := concat(str1:=WelcomeMessage, STR2:= concat(str1:=
	ParamSeparateur, str2:=concat(STR1:=ForDay, STR2:=concat(str1:= ParamSeparateur, STR2:= concat(str1:= 
	CalDate,str2:=concat(str1:= ParamSeparateur, str2 := CONCAT(str1:=
	ForPlant,str2:=Concat(str1:=ParamSeparateur, str2:= CONCAT(str1:= GetHostName.sHostName, str2:=ParamSeparateur)))))))));

IF InitLine <> LastInitLine OR InitLine = '' THEN
	LastInitLine := InitLine;
	bInitWriting := TRUE;
END_IF
	
IF FUN_CreateDir_CSV.bDirOK THEN
	FindFile
	(
		sNetId := '',
		sPathName := concat(FUN_CreateDir_CSV.AX_DirNames[2],CalFileName),
		eCmd := eEnumCmd_First,
		bExecute := TRUE,
		tTimeout := T#3S,
		stFindFile => FileInfo
	);
	
MesData.TimeCreation 	:= FILETIME_TO_SYSTEMTIME(filetime := FileInfo.creationTime);
MesData.TimeModif	 	:= FILETIME_TO_SYSTEMTIME(filetime := FileInfo.lastWriteTime);
MesData.FileSize  		:= ULARGE_TO_ULINT(in := FileInfo.fileSize);	
	
	IF NOT FindFile.bBusy THEN
		FindFile(bExecute := FALSE);
		bFileOK := MesData.FileSize > 0 ; 
	END_IF
	
	IF FindFile.bError OR  NOT bFileOK THEN
		FUN_CreateDir_CSV(InDirectory := ParamDirBaseStore, RESET2 := TRUE);
	END_IF
	
	IF NOT FindFile.bBusy AND NOT bFileOK AND bInitWriting THEN
		// je réinitialise les longueurs
		len_to_write := 0;
		MessageInitial := MessageInitialNull;
		MEMCPY(destAddr := ADR(MessageInitial)+len_to_write, srcAddr := ADR(InitLine), n := len(InitLine));
		len_to_add := len(InitLine);			len_to_write := len_to_write + len_to_add;
		
		MEMCPY(destAddr := ADR(MessageInitial)+len_to_write, srcAddr := ADR(NewLineVar), n := len(NewLineVar));
		len_to_add := len(NewLineVar);			len_to_write := len_to_write + len_to_add;
		
		MEMCPY(destAddr := ADR(MessageInitial)+len_to_write, srcAddr := ADR(TimeStampVar), n := len(TimeStampVar));
		len_to_add := len(TimeStampVar);		len_to_write := len_to_write + len_to_add;
		
		MEMCPY(destAddr := ADR(MessageInitial)+len_to_write, srcAddr := ADR(ParamSeparateur), n := len(ParamSeparateur));
		len_to_add := len(ParamSeparateur);		len_to_write := len_to_write + len_to_add;
		
		FOR KK := 1 TO ParamNbColumns DO
			MEMCPY(destAddr := ADR(MessageInitial)+len_to_write, srcAddr := ADR(AX_StructureValues[KK].Description), n := len(AX_StructureValues[KK].Description));
			len_to_add := len(AX_StructureValues[KK].Description);			len_to_write := len_to_write + len_to_add;
			
			MEMCPY(destAddr := ADR(MessageInitial)+len_to_write, srcAddr := ADR(ParamSeparateur), n := len(ParamSeparateur));
			len_to_add := len(ParamSeparateur);								len_to_write := len_to_write + len_to_add;
		END_FOR
		
		MEMCPY(destAddr := ADR(MessageInitial)+len_to_write, srcAddr := ADR(NewLineVar), n := len(NewLineVar));
		len_to_add := len(NewLineVar);			len_to_write := len_to_write + len_to_add;
		
		WriteFileInit
		(
			InStart := TRUE,
			InDirFile := concat(FUN_CreateDir_CSV.AX_DirNames[2], CalFileName),
			InAmsId := '', 
			InPMessage := ADR(MessageInitial),
			InLMessage := len_to_write
		);
		
		IF WriteFileInit.OutCompleted THEN
			WriteFileInit(InStart := FALSE);
			bInitWriting := FALSE;
		END_IF
	END_IF
	
	
	// Write file on SampleRate
	
	TriggerSampling(clk := CalLocalTimeStruct.wSecond = 10);

	IF bFileOK AND MesData.FileSize < 100000000 AND NOT bInitWriting   THEN
		len_to_write := 0;
		LineToWrite := LineToWrite_Null;
		MEMCPY(destAddr := ADR(LineToWrite)+len_to_write, srcAddr := ADR(MesTimeStamp), n := len(MesTimeStamp));
		len_to_add := len(MesTimeStamp);		len_to_write := len_to_write + len_to_add;
		
		MEMCPY(destAddr := ADR(LineToWrite)+len_to_write, srcAddr := ADR(ParamSeparateur), n := len(ParamSeparateur));
		len_to_add := len(ParamSeparateur);		len_to_write := len_to_write + len_to_add;
		
		FOR KK := 1 TO ParamNbColumns DO
			ReplaceAll(IN_StringToSearch := REAL_TO_STRING(AX_AverageValues[KK]), IN_StringToFind := '.', IN_StringToReplace := ParamDec, OUT_StringToSearch => ValueToWrite);
			//ValueToWrite := REAL_TO_STRING(AX_AverageValues[KK]);
			MEMCPY(destAddr := ADR(LineToWrite)+len_to_write, srcAddr := ADR(ValueToWrite), n := len(ValueToWrite));
			len_to_add := len(ValueToWrite);	len_to_write := len_to_write + len_to_add;
			
			MEMCPY(destAddr := ADR(LineToWrite)+len_to_write, srcAddr := ADR(ParamSeparateur), n := len(ParamSeparateur));
			len_to_add := len(ParamSeparateur);	len_to_write := len_to_write + len_to_add;
		END_FOR
		MEMCPY(destAddr := ADR(LineToWrite)+len_to_write, srcAddr := ADR(NewLineVar), n := len(NewLineVar));
		len_to_add := len(NewLineVar);			len_to_write := len_to_write + len_to_add;
		
		WriteFile
		(
			InStart := TriggerSampling.Q,
			InDirFile := concat(FUN_CreateDir_CSV.AX_DirNames[2], CalFileName),
			InAmsId := '', 
			InpMessage := ADR(LineToWrite),
			InLMessage := len_to_write
		);
		
		IF NOT WriteFile.OutBusy AND NOT WriteFile.OutError AND WriteFile.OutCompleted THEN
			// File has been writen successfully
			bWriteAlarm	:= FALSE ;
		ELSIF WriteFile.OutError THEN 
			// In case of writing error, try again to write the alarm. 
			bWriteAlarm	:= TRUE ;
		
		END_IF		
		
		
		
		
		
		
	END_IF

END_IF

CompressFile(IN_Directory := InDirectory);

METHOD M_AlarmManager
VAR

	FB_AlarmCodeManager			: FB_AlarmCodeManager ;

END_VAR
TON_WritealarmFile(IN:= NOT bFileOK  , PT:= T#10S  ) ;

// ALARM CODE //
	FB_AlarmCodeManager(
		bAlarm1			:= bWriteAlarm	  ,				// Write CSV Alarm
		bAlarm2			:= FALSE   ,					// 
		bAlarm3			:= TON_WritealarmFile.Q   ,		// Can not create CSV Alarm file 
		bAlarm4			:= FALSE	 ,					//
		bAlarm5			:= FALSE	,					// 
		bAlarm6			:= FALSE,									//
		bAlarm7			:= FALSE,                                   //
		bAlarm8			:= FALSE,                                   //
		bAlarm9			:= FALSE,                                   //
		bAlarm10		:= FALSE,                                   //
		bAlarm11		:= FALSE,									//
		bAlarm12		:= FALSE,                                   //
		bAlarm13		:= FALSE,                                   //
		bAlarm14		:= FALSE,                                   //
		bAlarm15		:= FALSE,                                   //
		wAlarmCode		=>MesData.MesAlarmCode);
END_METHOD

METHOD M_DataProcessing : BOOL
VAR
		
	KK : UINT;
END_VAR
FOR KK := 1 TO ParamNbColumns DO 
	IF AX_StructureValues[KK].Address <> 0 THEN 	
		AX_AverageFunctions[KK](ValueIn := AX_StructureValues[KK].Address^, WindowDuration := AX_StructureValues[KK].Sampling, ValueOut=> AX_AverageValues[KK]);	
	ELSIF AX_StructureValues[KK].AddressLR <> 0 THEN 	
		AX_AverageFunctions[KK](ValueIn := AX_StructureValues[KK].AddressLR^, WindowDuration := AX_StructureValues[KK].Sampling, ValueOut=> AX_AverageValues[KK]);	
	ELSIF AX_StructureValues[KK].AddressUL <> 0 THEN 	
		AX_AverageFunctions[KK](ValueIn := AX_StructureValues[KK].AddressUL^, WindowDuration := AX_StructureValues[KK].Sampling, ValueOut=> AX_AverageValues[KK]);	
	ELSIF AX_StructureValues[KK].AddressUI <> 0 THEN
		AX_AverageFunctions[KK](ValueIn := AX_StructureValues[KK].AddressUI^, WindowDuration := AX_StructureValues[KK].Sampling, ValueOut=> AX_AverageValues[KK]);			
	ELSE
		AX_AverageValues[KK] := 0;
	END_IF
END_FOR
END_METHOD

END_FUNCTION_BLOCK

// ---- 00_FunctionsBlocks/Fifo/FB_CommandAlternate.TcPOU
FUNCTION_BLOCK FB_CommandAlternate
VAR_INPUT
	AX_CMD 			: ARRAY[1..6] OF INV_Cmd;
	In_NB_Prio		: UINT;							
	ParamNbCMD		: UINT := 6;					// Number of elements of AX_CMD array
	In_Pulse		: BOOL;
END_VAR

VAR_OUTPUT
	CmdOutput		: INV_Cmd	;
END_VAR
VAR
	LastPosition 	: UINT;
	KK				: UINT;
	bInterrupt		: BOOL;
	Debut			: UINT;
	Fin				: UINT;
	Trig_Detec		: R_TRIG;
END_VAR

bInterrupt := FALSE;
Trig_Detec(CLK := In_Pulse);

IF Trig_Detec.Q THEN
	FOR KK := 1 TO In_NB_Prio DO
		IF AX_CMD[KK].bCmdStart^ THEN
			bInterrupt 	:= TRUE;
			CmdOutput := AX_CMD[KK];
			EXIT;
		END_IF
	END_FOR
	
	IF NOT bInterrupt THEN
		Debut := MAX(In_NB_Prio + 1, LastPosition + 1);
		Fin := Debut + ParamNbCMD - In_NB_Prio - 1;
		FOR KK := Debut TO Fin DO
			IF AX_CMD[KK - BOOL_TO_UINT(KK > ParamNbCMD)*(Fin - Debut + 1)].bCmdStart^ THEN
				LastPosition := KK - BOOL_TO_UINT(KK > ParamNbCMD)*(Fin - Debut + 1);
				CmdOutput := AX_CMD[ KK - BOOL_TO_UINT(KK > ParamNbCMD)*(Fin - Debut + 1)];
				EXIT ;
			END_IF
		END_FOR
	END_IF
END_IF

END_FUNCTION_BLOCK

// ---- 00_FunctionsBlocks/HistorizationVisu/FB_OperationIndex.TcPOU
FUNCTION_BLOCK FB_OperationIndex
////////////////// 
// Get Operationnal Indicators . Number of movements. Running hours, Last Move datetime 
//////////////////	
VAR_INPUT
	MesON				: BOOL ; 
	CmdReset			: BOOL ;

END_VAR

VAR_OUTPUT PERSISTENT
	CalRunningTimeHr	: INT ; 	// (Hrs) Running Time  
	CalNbMove			: WORD ;
	CalTimeStart		: STRING 	;	// DateTime at last Move .  ( hour Granularity ) .

END_VAR

VAR PERSISTENT
	CalRunningTime		: TIME ;
	CalRunningTime_Temp	: TIME;		// Previous RunningTime ater last move. 
	CTU 				: CTU ;		// Count the nb of moves 
	
END_VAR 

VAR 
	ElapsedTime 		: TIME ;	//  Elapsed Time since last move 
	CurrentTime 		: TIME ; 	// Current Time 
	TimeStart			: TIME 	;	// TImeHour when the Move starts for the last time
	R_TRIG 				: R_TRIG ; 	// Detect move starts
	F_TRIG 				: F_TRIG ; 	// Detect move stops

END_VAR


// RESET //
	IF CmdReset THEN 
		TimeStart 			:= TIME() ; 
		CalRunningTime 		:= T#0MS ; 
		CalRunningTime_Temp := T#0MS ;
		CTU(CU:=FALSE) ; 
		CTU(RESET:=TRUE); 
	END_IF



// NUMBER OF MOVES //
//	CTU(CU := MesON , RESET:=FALSE , PV:=65535 , CV => CalNbMove ) ; 
	
// RUNNING HOURS //
	R_TRIG(CLK:= MesON ) ; 
	F_TRIG(CLK:= MesON ) ; 
	
	CurrentTime := TIME() ;
	
	IF R_TRIG.Q THEN 
		TimeStart := TIME() ; 
		CalTimeStart := LEFT(sTimeLocal_G, 16);	 // Minutes granularity . 
	END_IF
	
	ElapsedTime 	:= CurrentTime - TimeStart ;	
	IF MesON THEN 
 
		CalRunningTime  := CalRunningTime_Temp +  ElapsedTime ;
		
	ELSE
		CalRunningTime_Temp := CalRunningTime ; 
		
	END_IF

	CalRunningTimeHr	:= DWORD_TO_INT(TIME_TO_DWORD(CalRunningTime)/1000/3600) ;

END_FUNCTION_BLOCK

// ---- 00_FunctionsBlocks/HistorizationVisu/GetTime.TcPOU
PROGRAM GetTime
VAR
	
	// DATETIME //
		FB_GetSystemTime        : GETSYSTEMTIME;
		FB_ToLocal 				: FB_FileTimeToTzSpecificLocalTime;
		fileTime        		: T_FILETIME;
		FileTimeLocal			: T_FILETIME;
	
	//TEST//
		VarTest AT %I* 			: UINT ; 		// Test variable to be linked to ethercat devices before activation to run tests without complete powerplant.
	
END_VAR

	// DateTime 
	FB_GetSystemTime(
		timeLoDW	=> fileTime.dwLowDateTime, 
		timeHiDW	=> fileTime.dwHighDateTime);
		
	FB_ToLocal(
		in			:=fileTime,
		tzInfo 		:= CstTimeZone_G,
		out		 	=> FileTimeLocal);
		
	sTimeGMT_G 		:= SYSTEMTIME_TO_STRING(FILETIME_TO_SYSTEMTIME(fileTime));	// Full Date Time with ms granularity GMT
	sTimeLocal_G	:= SYSTEMTIME_TO_STRING (FILETIME_TO_SYSTEMTIME(FileTimeLocal));

END_PROGRAM

// ---- 00_FunctionsBlocks/Templates/FB_EX_Example.TcPOU
FUNCTION_BLOCK FB_EX_Example
//////////////////
// 
//////////////////
VAR CONSTANT PERSISTENT
	// Characteristics of the object (Same for all instances)
	
END_VAR

VAR_INPUT PERSISTENT
	// Parameters of the Object (instance specific) 
	
END_VAR

VAR_OUTPUT
	//Child objects
	
END_VAR
VAR
	//M_METHOD2 VARIABLES//
	
	
	//M_METHOD2 VARIABLES//
	
	
	//M_METHOD3 VARIABLES//
	
	
	//GET/SET PROPERTY MANAGEMENT//
	
	
END_VAR

END_FUNCTION_BLOCK

// ---- 01_Equipement_Library/Actuators/FB_CB_AuxMVCB.TcPOU
FUNCTION_BLOCK FB_CB_AuxMVCB EXTENDS FB_CB_Base
//////////////////
//  Motorized Circuit Breaker with telecommAND   Requires Open and Close impulsions.
//////////////////

VAR_INPUT PERSISTENT
	// Parameters of the Object (instance/model specific) 
	ParamTP_Impulsion	   : TIME := T#2S ;			// (s) 	 Config : Tempo for the start or stop command impulsion
	ParamFuseNC		       : BOOL ;					//  False: TRUE = Closed , True : TRUE = opened	
END_VAR

VAR_OUTPUT
	//Child objects
	
END_VAR

VAR_INPUT
	// I/O Inputs              
	IN_MesFuse_IO				: BOOL;
	IN_MesEarth_IO			: BOOL ; 
	
END_VAR

VAR
	//M_OPENCLOSE VARIABLES//	
		RsFuse			:RS ;
		
	//M_ALARMMANAGEMENT VARIABLES//
	MesDataExd	: CB_AuxMVCB_Sch;
 
	//M_STATEMANAGER VARIABLES//
	
	// M_EXECUTE VARIABLES //
		
 
END_VAR

METHOD M_Execute
VAR_INPUT
END_VAR



SUPER^.M_Execute();
// updat.MesDataExd.MesData.to be used in other functions 
MesDataExd.MesData.MesClosed := RS_Emulate.Q1 ;
END_METHOD

END_FUNCTION_BLOCK

// ---- 01_Equipement_Library/Actuators/FB_CB_Base.TcPOU
FUNCTION_BLOCK FB_CB_Base
//////////////////
// Electrical Switch - Base FB
//////////////////
VAR_INPUT
	// Parameters of the Object (instance specific) 
	IN_CmdExternalOpen_Emul			: BOOL ; 
	IN_CmdExternalClose_Emul		: BOOL ;
	
END_VAR
VAR
	bInit							: BOOL := TRUE ;

	TON_OutputWait_Open				: TON;
	TON_OutputWait_Close			: TON;
	
	ParamTimeOpen_Wait				: TIME := T#1S;
	ParamTimeClose_Wait				: TIME := T#1S;
	RS_Emulate: RS;
	R_TRIGOpen: R_TRIG;
	R_TRIGClose: R_TRIG;
	
END_VAR
VAR_INPUT PERSISTENT
	// Parameters of the Object (instance/model specific) 
	ParamTimeOut_Open       		: TIME  := T#1S     ;       // (ms) Config : Tempo to open before Timeout warning  
	ParamTimeOut_Close      		: TIME  := T#1S     ;		// (ms) Config : Tempo to close before Timeout warning
	ParamTimeOut_Alarm   		    : TIME  := T#200MS  ;		// (ms) Config : Tempo when open and close before raising alarm // Check tag, original : ParamTempoStateAlarm
	ParamNC							: BOOL  := FALSE    ;		// (NA) False: TRUE = Closed , True : TRUE = opened             // Check description
	ParamNbFdbck			    	: BYTE              ;		// (NA) Number of Feedback Position (1: 1 wire , 2 : 2 wire)    // Check tag
	ParamClosedInput_Connected		: BOOL  := TRUE     ; 		// (NA)True : closed input is connected                         // Check tag
	                                                    	
END_VAR

VAR_OUTPUT
	//Child objects
	
END_VAR

VAR_INPUT
	// I/O Inputs 
		IN_MesOpened_IO					: BOOL  ; 				// (NA) [P,H,B] Opened Position IO	         //Check: MesOpened is another var 
		IN_MesClosed_IO 				: BOOL := TRUE ; 		// (NA) [P,H,B] Closed Position IO           //Check: MesClosed is another var
	
		IN_CmdOpen 						: BOOL ; 				// (NA) External Open Command 
		IN_CmdClose						: BOOL ; 				// (NA) External Close Command 
		IN_CmdReset_L					: BOOL ;				// (NA) External Reset Command              // Check: what does the L respresent ? 
		
END_VAR

VAR
	//M_OPENCLOSE VARIABLES//
		MesOpened					     : BOOL ;                                                                     //Check: MesClosed is another var
		MesClosed					     : BOOL ;                                                                     //Check: MesOpened is another var
		
	//M_ALARMMANAGEMENT VARIABLES//
		FB_CheckCommand				     : FB_CheckCommand ; 	//(NA) Check if start command successful 
		FB_CheckCommand2			     : FB_CheckCommand ;		//(NA) Check if stop command successful  
		TON_ClosedAndOpened			     : TON ;              	
		TON_NotClosedAndNotOpened	     : TON ;              	
                                             	
		
		
	//M_STATEMANAGER VARIABLES//
		MesState					     : BYTE ; 				// (NA) Cal [P,H,B] Bit 0: Open , Bit 1: Closed        // Check : Cal ? BYTE or BOOL ?
	///MesDataExd				     : CB ; 

	// M_EXECUTE VARIABLES 	//                                   


		
END_VAR

METHOD M_Execute
VAR_INPUT
END_VAR
RS_Emulate(SET := MesClosed OR IN_CmdExternalClose_Emul , RESET1 := MesOpened OR IN_CmdExternalOpen_Emul ); 			// The Cell opens after receiving a open order or if receiving an external open ordre ( C13100 , .. ) 



IF ParamNC THEN 
	IN_MesOpened_IO 		:= RS_Emulate.Q1 ;  						// CB Opened if CmdOpenedIO
	IN_MesClosed_IO 		:= NOT RS_Emulate.Q1 ; 								// Cb Closed if CmdClosedIO
ELSE 
	IN_MesOpened_IO 		:= NOT RS_Emulate.Q1 ;  						// CB Opened if CmdOpenedIO
	IN_MesClosed_IO 		:= RS_Emulate.Q1 ; 								// Cb Closed if CmdClosedIO
END_IF

R_TRIGOpen(CLK:= IN_MesOpened_IO AND NOT bInit ) ; 
R_TRIGClose(CLK:= IN_MesClosed_IO AND NOT bInit  ) ; // do not write on the first cycle time ( to allow emul variable to be set from outside)

IF bInit THEN 
	bInit := FALSE ; 
END_IF
END_METHOD

END_FUNCTION_BLOCK

// ---- 01_Equipement_Library/Actuators/FB_CB_FeederMVCB.TcPOU
FUNCTION_BLOCK FB_CB_FeederMVCB EXTENDS FB_CB_Base
//////////////////
//  Motorized Circuit Breaker with telecommAND   Requires Open and Close impulsions.
//////////////////


VAR_INPUT PERSISTENT
	// Parameters of the Object (instance/model specific) 
	ParamTP_Impulsion		    : TIME 		:= T#2S ;	// (s) Config : Tempo for the start or stop command impulsion
	ParamComutNc			    : BOOL ;				// Local selector in normally closed . NC >> True = Selector in local. 
	ParamSectLigne			    : BYTE      :=1 ;		// Monitoring du sectionneur de ligne de la MainMVCB .0 = TRUE := Monitoré .1 = TRUE Close is connected

END_VAR
VAR_INPUT
	A1_Sect				       : FB_CB_MVSwitch;

// I/O Inputs              
	IN_MesAlarmPwr_IO		           : BOOL ;	              // (NA)[P,H,B] Remote control Power supply Error .  IO  	
	IN_MesTripped_IO		  		   : BOOL ; 	          // Tripped position of the CB Must Ack To switch in again
	IN_MesComutLocal_IO			   	   : BOOL := TRUE ; 	  // True if cell is in local position . 
	IN_MesEarth_IO 			       : BOOL ; 	
		
END_VAR
VAR_OUTPUT 
	OUT_CmdOpen_IO	          	   : BOOL ; 	          // (NA) Physical I/O Open Command IO
	OUT_CmdClose_IO			   : BOOL ; 	          // (NA) Physical I/O Close Command IO
END_VAR

VAR
	//M_OPENCLOSE VARIABLES//
	MesDataExd					: CB_FeederMVCB_Sch ; 
	
	//M_ALARMMANAGEMENT VARIABLES//
		
	//M_STATEMANAGER VARIABLES//
	
	// M_EXECUTE VARIABLES //
		
	// EMULATOR //

		
END_VAR

METHOD M_Execute
VAR_INPUT
END_VAR

VAR

END_VAR


TON_OutputWait_Open(IN := OUT_CmdOpen_IO, PT := ParamTimeOpen_Wait, Q => MesOpened);
TON_OutputWait_Close(IN :=OUT_CmdClose_IO, PT := ParamTimeClose_Wait, Q => MesClosed);



SUPER^.M_Execute();

// updat.MesDataExd.MesData.to be used in other functions 
MesDataExd.MesData.MesClosed := RS_Emulate.Q1 ;
END_METHOD

END_FUNCTION_BLOCK

// ---- 01_Equipement_Library/Actuators/FB_CB_MVSwitch.TcPOU
FUNCTION_BLOCK FB_CB_MVSwitch EXTENDS FB_CB_Base
//////////////////
//  Motorized Circuit Breaker with telecommAND   Requires Open and Close impulsions.
//////////////////

VAR_INPUT PERSISTENT
	// Parameters of the Object (instance/model specific) 
	
END_VAR

VAR_INPUT
	// I/O Inputs              	
		
END_VAR

VAR
	//M_OPENCLOSE VARIABLES//

	
	//M_ALARMMANAGEMENT VARIABLES//
		
	//M_STATEMANAGER VARIABLES//
MesDataExd	       			 :  CB_Standard ; 
	// M_EXECUTE VARIABLES //
		
	// EMULATOR //

		
END_VAR

METHOD M_Execute
VAR_INPUT
END_VAR



SUPER^.M_Execute();

// updat.MesDataExd.MesData.to be used in other functions 
MesDataExd.MesData.MesClosed := RS_Emulate.Q1 ;
END_METHOD

END_FUNCTION_BLOCK

// ---- 01_Equipement_Library/Actuators/FB_CB_GridMVCB.TcPOU
FUNCTION_BLOCK FB_CB_GridMVCB EXTENDS FB_CB_Base
//////////////////
//  Motorized Circuit Breaker with telecommAND   Requires Open and Close impulsions.
//////////////////

VAR_INPUT PERSISTENT
	// Parameters of the Object (instance/model specific) 
	
END_VAR

VAR_INPUT
	// I/O Inputs              	
		
END_VAR

VAR
	//M_OPENCLOSE VARIABLES//

	
	//M_ALARMMANAGEMENT VARIABLES//
		
	//M_STATEMANAGER VARIABLES//
MesDataExd			: CB_Standard ; 
	// M_EXECUTE VARIABLES //
		
	// EMULATOR //

		
END_VAR

METHOD M_Execute
VAR_INPUT
END_VAR



SUPER^.M_Execute();

// updat.MesDataExd.MesData.to be used in other functions 
MesDataExd.MesData.MesClosed := RS_Emulate.Q1 ;
END_METHOD

END_FUNCTION_BLOCK

// ---- 01_Equipement_Library/Actuators/FB_CB_MainHVCB.TcPOU
FUNCTION_BLOCK FB_CB_MainHVCB EXTENDS FB_CB_Base
//////////////////
//  Motorized Circuit Breaker with telecommAND  Requires Open and Close impulsions.
//////////////////

VAR_INPUT PERSISTENT
	// Parameters of the Object (instance/model specific) 
	ParamTP_Impulsion		    : TIME 		:= T#2S ;	// (s) Config : Tempo for the start or stop command impulsion
	ParamComutNc			    : BOOL ;
	ParamSectLigne			    : BYTE      :=1 ;		// Monitoring du sectionneur de ligne de la MainMVCB .0 = TRUE := Monitoré .1 = TRUE Close is connected

END_VAR

VAR_OUTPUT
	//Child objects
	
END_VAR

VAR_INPUT
	A1_Sect				       : FB_CB_MVSwitch;

// I/O Inputs              
	IN_MesAlarmPwr_IO		           : BOOL ;	              // (NA)[P,H,B] Remote control Power supply Error .  IO  	
	IN_MesTripped_IO		  		   : BOOL ; 	          // Tripped position of the CB Must Ack To switch in again
	IN_MesComut_IO			   	   : BOOL := TRUE ; 	  // True if cell is in local position . 
	IN_MesEarth_IO 			       : BOOL ; 	
		
END_VAR

VAR
	//M_OPENCLOSE VARIABLES//	
	TP_Open	 			: TP ;				// (NA) Temporisation for Open pulse Command
	TP_Close 				: TP ;				// (NA) Temporisation for Close pulse Command	

	//M_ALARMMANAGEMENT VARIABLES//
MesDataExd	        :  CB_MainHVCB_Sch ; 
	
//M_STATEMANAGER VARIABLES//
	
END_VAR

METHOD M_Execute
VAR_INPUT
END_VAR

VAR

END_VAR

SUPER^.M_Execute();

// updat.MesDataExd.MesData.to be used in other functions 
MesDataExd.MesData.MesClosed := RS_Emulate.Q1 ;
END_METHOD

END_FUNCTION_BLOCK

// ---- 01_Equipement_Library/Actuators/FB_CB_MainMVCB.TcPOU
FUNCTION_BLOCK FB_CB_MainMVCB EXTENDS FB_CB_Base
//////////////////
//  Motorized Circuit Breaker with telecommAND  Requires Open and Close impulsions.
//////////////////

VAR_INPUT PERSISTENT
	// Parameters of the Object (instance/model specific) 
	ParamTP_Impulsion		    : TIME 		:= T#2S ;	// (s) Config : Tempo for the start or stop command impulsion
	ParamComutNc			    : BOOL ;				// Local selector in normally closed . NC >> True = Selector in local. 
	ParamSectLigne			    : BYTE      :=1 ;		// Monitoring du sectionneur de ligne de la MainMVCB .0 = TRUE := Monitoré .1 = TRUE Close is connected

END_VAR

VAR_OUTPUT
	//Child objects
	OUT_CmdOpen_IO	          	   : BOOL ; 	          // (NA) Physical I/O Open Command IO
	OUT_CmdClose_IO			   : BOOL ; 	          // (NA) Physical I/O Close Command IO
	
END_VAR

VAR_INPUT
	A1_Sect				        : FB_CB_MVSwitch;

// I/O Inputs              
	IN_MesAlarmPwr_IO		           : BOOL ;	              // (NA)[P,H,B] Remote control Power supply Error .  IO  	
	IN_MesTripped_IO		  		   : BOOL ; 	          // Tripped position of the CB Must Ack To switch in again
	IN_MesComutLocal_IO			   	   : BOOL := TRUE ; 	  // True if cell is in local position . 
	IN_MesEarth_IO 			       : BOOL ; 	
		
END_VAR

VAR
	//M_OPENCLOSE VARIABLES//	
	ParamTP_Open	 			: TP ;				// (NA) Temporisation for Open pulse Command
	ParamTP_Close 				: TP ;				// (NA) Temporisation for Close pulse Command	

	//M_ALARMMANAGEMENT VARIABLES//
MesDataExd	        :  CB_MainMVCB_Sch ; 
	
//M_STATEMANAGER VARIABLES//
	
END_VAR

METHOD M_Execute
VAR_INPUT
END_VAR

VAR

END_VAR
TON_OutputWait_Open(IN := OUT_CmdOpen_IO, PT := ParamTimeOpen_Wait, Q => MesOpened);
TON_OutputWait_Close(IN :=OUT_CmdClose_IO, PT := ParamTimeClose_Wait, Q => MesClosed);

IF ParamSectLigne.0 THEN 
	A1_Sect.M_Execute();
END_IF

SUPER^.M_Execute();
// updat.MesDataExd.MesData.to be used in other functions 
MesDataExd.MesData.MesClosed := RS_Emulate.Q1 ;
END_METHOD

END_FUNCTION_BLOCK

// ---- 01_Equipement_Library/Actuators/FB_CB_MeasureMVCB.TcPOU
FUNCTION_BLOCK FB_CB_MeasureMVCB EXTENDS FB_CB_Base
//////////////////
//  Motorized Circuit Breaker with telecommAND   Requires Open and Close impulsions.
//////////////////

VAR_INPUT PERSISTENT
	// Parameters of the Object (instance/model specific) 
	ParamTP_Impulsion	   : TIME := T#2S ;			// (s) 	 Config : Tempo for the start or stop command impulsion
	ParamFuseNC		       : BOOL ;					//  False: TRUE = Closed , True : TRUE = opened	
END_VAR

VAR_OUTPUT
	//Child objects
	
END_VAR

VAR_INPUT
	// I/O Inputs              
	IN_MesFuse_IO				: BOOL;
	IN_MesEarth_IO			: BOOL ; 
	
END_VAR

VAR
	//M_OPENCLOSE VARIABLES//	
		RsFuse			:RS ;
		
	//M_ALARMMANAGEMENT VARIABLES//
	MesDataExd	: CB_MeasureMVCB_Sch ;
 
	//M_STATEMANAGER VARIABLES//
	
	// M_EXECUTE VARIABLES //
		
 
END_VAR

METHOD M_Execute
VAR_INPUT
END_VAR



SUPER^.M_Execute();

// updat.MesDataExd.MesData.to be used in other functions 
MesDataExd.MesData.MesClosed := RS_Emulate.Q1 ;
END_METHOD

END_FUNCTION_BLOCK

// ---- 01_Equipement_Library/Batteries/FB_SystemBMS_Base.TcPOU
FUNCTION_BLOCK FB_SystemBMS_Base

VAR_INPUT PERSISTENT
	// Parameters of the Object (instance specific) 
	ParamTempoComAlarm			: TIME 		:= T#10S ; 				// (s) Config : Tempo to detect LOC Alarm
	ParamTimeOutStart           : TIME 		:= T#60S ;				// (s) Config : Tempo to start before Timeout warning
	ParamTimeOutStop        	: TIME 		:= T#5S ;				// (s) Config : Tempo to start before Timeout warning

	ParamEnomRack				: REAL 	:= 97.2 ;  	  	// (kWh) Nominal Energy Capacity of one Rack 
	
	ParamClockReadTime 			: TIME := TIME#1S;	  				// (Time) Read Modbus Frequency .   
	ParamClockWriteTime 		: TIME := TIME#1S;   			// (Time) Write Modbus Frequency .         
	ParamTimeout				: TIME  := T#1S ;		  			// (Time) Timeout for modbus reading
	ParamTimeWatchdog			: TIME := T#30S;						// (Time) Time after which a fixed watchdog raises an alarm
	
	
	ParamNbRacks				: BYTE 	:= 17 ; 					// (NA) Number of racks controlled .
	ParamEssNum					: UINT := 1;						// (NA) ID number of the SystemBms' father PCS
	ParamSystemBmsNum			: UINT := 1;						// Ctrl Bat Index in case of several CtrlBat 						
	

	
	
END_VAR

VAR_INPUT
	//Child objects
	  
END_VAR

VAR
	//M_ALARMMANAGEMENT VARIABLES//

	MesDataExd				AT%Q* : SystemBMS ;											// (NA) [P,H,B] CTRLbat  Data Structure
	
	
		ClockRead				AT %Q*		: BOOL;							// (NA) Modbus reading Clock
		ClockWrite 				AT %Q*		: BOOL;							// (NA) Modbus writing Clock 	
		
	//M_INIT VARIABLES //
		bInit						: BOOL 				:= TRUE ; 		// (NA) Initialize object parameters at first cycle 
		

END_VAR

METHOD M_Evaluate : BOOL
VAR_INPUT
END_VAR
END_METHOD

METHOD M_Execute
//////////////////
//  Method Calls 
/////////////////

VAR 
	// Method local variables (reinitialized at each cycle) 
	KK		: INT;

	MesModbusReadAlarm: INT;
END_VAR
// READING AND WRITING CLOCK //
	TP1(IN:=NOT TP1.Q , PT:= ParamClockReadTime);
	ClockRead 	:= TP1.Q ;
	
	TP2(IN:=NOT TP2.Q , PT:= ParamClockWriteTime);
	ClockWrite 	:= TP2.Q;	
	
// PERMANENT CONDITIONS //
	M_CP() ; 

